   A_3126_BTE05.Par.OutDelayTime := 0;
   A_3126_BTE05.Par.Spare66 := 0;
   A_3126_BTE06.StCode := 0;
   A_3126_BTE06.InMonLL := FALSE;
   A_3126_BTE06.InMonL := FALSE;
   A_3126_BTE06.InMonMid := FALSE;
   A_3126_BTE06.InMonH := FALSE;
   A_3126_BTE06.InMonHH := FALSE;
   A_3126_BTE06.spare0205 := FALSE;
   A_3126_BTE06.InpFaultAI := FALSE;
   A_3126_BTE06.InpFaultDev := FALSE;
   A_3126_BTE06.InHWStop := FALSE;
   A_3126_BTE06.InDPFault := FALSE;
   A_3126_BTE06.InDisable := FALSE;
   A_3126_BTE06.CmdFaultReset := FALSE;
   A_3126_BTE06.InLocal := FALSE;
   A_3126_BTE06.spare0305 := FALSE;
   A_3126_BTE06.InReport := FALSE;
   A_3126_BTE06.spare0307 := FALSE;
   A_3126_BTE06.OutLL := FALSE;
   A_3126_BTE06.OutL := FALSE;
   A_3126_BTE06.OutH := FALSE;
   A_3126_BTE06.OutHH := FALSE;
   A_3126_BTE06.OutOverflow := FALSE;
   A_3126_BTE06.spare0405 := FALSE;
   A_3126_BTE06.OutFaultAI := FALSE;
   A_3126_BTE06.spare0407 := FALSE;
   A_3126_BTE06.StLL := FALSE;
   A_3126_BTE06.StL := FALSE;
   A_3126_BTE06.StMid := FALSE;
   A_3126_BTE06.StH := FALSE;
   A_3126_BTE06.StHH := FALSE;
   A_3126_BTE06.StFaultAI := FALSE;
   A_3126_BTE06.OutWarning := FALSE;
   A_3126_BTE06.OutFaulted := FALSE;
   A_3126_BTE06.InpValue := 0;
   A_3126_BTE06.OutValuePc := 0;
   A_3126_BTE06.OutValueUnits := L#0;
   A_3126_BTE06.Msg.WarningDoneLL := FALSE;
   A_3126_BTE06.Msg.WarningDoneL := FALSE;
   A_3126_BTE06.Msg.WarningDoneMid := FALSE;
   A_3126_BTE06.Msg.WarningDoneH := FALSE;
   A_3126_BTE06.Msg.WarningDoneHH := FALSE;
   A_3126_BTE06.Msg.FaultDoneLL := FALSE;
   A_3126_BTE06.Msg.FaultDoneL := FALSE;
   A_3126_BTE06.Msg.FaultDoneMid := FALSE;
   A_3126_BTE06.Msg.FaultDoneH := FALSE;
   A_3126_BTE06.Msg.FaultDoneHH := FALSE;
   A_3126_BTE06.Msg.FaultDoneDev := FALSE;
   A_3126_BTE06.Msg.FaultDoneAI := FALSE;
   A_3126_BTE06.OutAlarmNrLog := 0;
   A_3126_BTE06.Par.ParObjectNo := 27118;
   A_3126_BTE06.Par.ParMsgType := 7252;
   A_3126_BTE06.Par.ParHornCode := 10;
   A_3126_BTE06.Par.ParLogOff := FALSE;
   A_3126_BTE06.Par.ParSpare0401 := FALSE;
   A_3126_BTE06.Par.ParValueByUser := FALSE;
   A_3126_BTE06.Par.ParLimitsPc := TRUE;
   A_3126_BTE06.Par.ParWago := FALSE;
   A_3126_BTE06.Par.ParNoHornByWarning := FALSE;
   A_3126_BTE06.Par.ParWarningLL := FALSE;
   A_3126_BTE06.Par.ParWarningL := FALSE;
   A_3126_BTE06.Par.ParWarningMid := FALSE;
   A_3126_BTE06.Par.ParWarningH := TRUE;
   A_3126_BTE06.Par.ParWarningHH := FALSE;
   A_3126_BTE06.Par.ParPreAlarmLL := FALSE;
   A_3126_BTE06.Par.ParPreAlarmL := FALSE;
   A_3126_BTE06.Par.ParPreAlarmMid := FALSE;
   A_3126_BTE06.Par.ParPreAlarmH := FALSE;
   A_3126_BTE06.Par.ParPreAlarmHH := FALSE;
   A_3126_BTE06.Par.ParUnitsByZeroDigit := L#0;
   A_3126_BTE06.Par.ParUnitsByMaxDigit := L#27384;
   A_3126_BTE06.Par.ParUnitsBy100Pc := L#10000;
   A_3126_BTE06.Par.ParLimitLL := L#0;
   A_3126_BTE06.Par.ParLimitL := L#2000;
   A_3126_BTE06.Par.ParLimitH := L#8000;
   A_3126_BTE06.Par.ParLimitHH := L#10000;
   A_3126_BTE06.Par.ParMonTimeLL := 0;
   A_3126_BTE06.Par.ParMonTimeL := 0;
   A_3126_BTE06.Par.ParMonTimeMid := 0;
   A_3126_BTE06.Par.ParMonTimeH := 600;
   A_3126_BTE06.Par.ParMonTimeHH := 0;
   A_3126_BTE06.Par.ParDelayTimeDown := 10;
   A_3126_BTE06.Par.ParDelayTimeUp := 10;
   A_3126_BTE06.Par.ParDelayTime := 30;
   A_3126_BTE06.Par.OutMonTimeLL := 0;
   A_3126_BTE06.Par.OutMonTimeL := 0;
   A_3126_BTE06.Par.OutMonTimeMid := 0;
   A_3126_BTE06.Par.OutMonTimeH := 0;
   A_3126_BTE06.Par.OutMonTimeHH := 0;
   A_3126_BTE06.Par.OutDelayTimeDown := 0;
   A_3126_BTE06.Par.OutDelayTimeUp := 0;
   A_3126_BTE06.Par.OutDelayTime := 0;
   A_3126_BTE06.Par.Spare66 := 0;
   A_3126_MXZ01MA.Ma.StCode := 0;
   A_3126_MXZ01MA.Ma.InEnableRev := FALSE;
   A_3126_MXZ01MA.Ma.InEnableFwd := FALSE;
   A_3126_MXZ01MA.Ma.InOverrideHLOutlet := FALSE;
   A_3126_MXZ01MA.Ma.spare0203 := FALSE;
   A_3126_MXZ01MA.Ma.OutEdgeFaultReset := FALSE;
   A_3126_MXZ01MA.Ma.OutFaultResetFcttst := FALSE;
   A_3126_MXZ01MA.Ma.InpControlEBM := FALSE;
   A_3126_MXZ01MA.Ma.InpLocked := FALSE;
   A_3126_MXZ01MA.Ma.CmdOff := FALSE;
   A_3126_MXZ01MA.Ma.CmdOn := FALSE;
   A_3126_MXZ01MA.Ma.CmdNext := FALSE;
   A_3126_MXZ01MA.Ma.CmdFaultReset := FALSE;
   A_3126_MXZ01MA.Ma.InLocal := FALSE;
   A_3126_MXZ01MA.Ma.InManual := FALSE;
   A_3126_MXZ01MA.Ma.CmdTestEBM := FALSE;
   A_3126_MXZ01MA.Ma.InSeqStop := FALSE;
   A_3126_MXZ01MA.Ma.OutWarning := FALSE;
   A_3126_MXZ01MA.Ma.InfBMTopOk := FALSE;
   A_3126_MXZ01MA.Ma.InfBMBottomOk := FALSE;
   A_3126_MXZ01MA.Ma.InfSMOk := FALSE;
   A_3126_MXZ01MA.Ma.OutpFcttst_BM_Top := FALSE;
   A_3126_MXZ01MA.Ma.OutpFcttst_BM_Bottom := FALSE;
   A_3126_MXZ01MA.Ma.OutpFcttst_SM := FALSE;
   A_3126_MXZ01MA.Ma.OutpFaultReset := FALSE;
   A_3126_MXZ01MA.Ma.StStopped := FALSE;
   A_3126_MXZ01MA.Ma.StStarting := FALSE;
   A_3126_MXZ01MA.Ma.StStartedFwd := FALSE;
   A_3126_MXZ01MA.Ma.StStopping := FALSE;
   A_3126_MXZ01MA.Ma.StFault := FALSE;
   A_3126_MXZ01MA.Ma.StStartedRev := FALSE;
   A_3126_MXZ01MA.Ma.StLocked := FALSE;
   A_3126_MXZ01MA.Ma.OutTestTime := 0;
   A_3126_MXZ01MA.Ma.Par.ParObjectNo := 27119;
   A_3126_MXZ01MA.Ma.Par.ParWithMon1 := TRUE;
   A_3126_MXZ01MA.Ma.Par.ParWithMon3 := FALSE;
   A_3126_MXZ01MA.Ma.Par.ParWithMon4 := TRUE;
   A_3126_MXZ01MA.Ma.Par.ParWithMon5 := FALSE;
   A_3126_MXZ01MA.Ma.Par.ParWithMon6 := FALSE;
   A_3126_MXZ01MA.Ma.Par.ParMon1IsHL := FALSE;
   A_3126_MXZ01MA.Ma.Par.ParMon1IsLS := TRUE;
   A_3126_MXZ01MA.Ma.Par.ParMon1StopByFault := TRUE;
   A_3126_MXZ01MA.Ma.Par.ParMon2IsLS := FALSE;
   A_3126_MXZ01MA.Ma.Par.ParMon3IsLS := FALSE;
   A_3126_MXZ01MA.Ma.Par.ParMon4AsWarning := FALSE;
   A_3126_MXZ01MA.Ma.Par.ParMon4StopByFault := FALSE;
   A_3126_MXZ01MA.Ma.Par.ParMon4IsLS := FALSE;
   A_3126_MXZ01MA.Ma.Par.ParEBM := FALSE;
   A_3126_MXZ01MA.Ma.Par.ParMon4IsSM := TRUE;
   A_3126_MXZ01MA.A_3126_KCU04.StCode := 0;
   A_3126_MXZ01MA.A_3126_KCU04.InMonTrue := FALSE;
   A_3126_MXZ01MA.A_3126_KCU04.InMonFalse := FALSE;
   A_3126_MXZ01MA.A_3126_KCU04.InPreAlarmTrue := FALSE;
   A_3126_MXZ01MA.A_3126_KCU04.InPreAlarmFalse := FALSE;
   A_3126_MXZ01MA.A_3126_KCU04.InStopTrueTime := FALSE;
   A_3126_MXZ01MA.A_3126_KCU04.InStopFalseTime := FALSE;
   A_3126_MXZ01MA.A_3126_KCU04.InpTrue := FALSE;
   A_3126_MXZ01MA.A_3126_KCU04.InpFaultDev := FALSE;
   A_3126_MXZ01MA.A_3126_KCU04.CmdRstTrueTime := FALSE;
   A_3126_MXZ01MA.A_3126_KCU04.CmdRstFalseTime := FALSE;
   A_3126_MXZ01MA.A_3126_KCU04.CmdRunTimeoutTime := FALSE;
   A_3126_MXZ01MA.A_3126_KCU04.CmdFaultReset := FALSE;
   A_3126_MXZ01MA.A_3126_KCU04.InLocal := FALSE;
   A_3126_MXZ01MA.A_3126_KCU04.spare0305 := FALSE;
   A_3126_MXZ01MA.A_3126_KCU04.InReport := FALSE;
   A_3126_MXZ01MA.A_3126_KCU04.OutTimeoutTime := FALSE;
   A_3126_MXZ01MA.A_3126_KCU04.InHWStop := FALSE;
   A_3126_MXZ01MA.A_3126_KCU04.InDPFault := FALSE;
   A_3126_MXZ01MA.A_3126_KCU04.OutPreAlarmTrue := FALSE;
   A_3126_MXZ01MA.A_3126_KCU04.OutPreAlarmFalse := FALSE;
   A_3126_MXZ01MA.A_3126_KCU04.OutFlagPos := FALSE;
   A_3126_MXZ01MA.A_3126_KCU04.OutFlagNeg := FALSE;
   A_3126_MXZ01MA.A_3126_KCU04.OutpFaultReset := FALSE;
   A_3126_MXZ01MA.A_3126_KCU04.OutTrue := FALSE;
   A_3126_MXZ01MA.A_3126_KCU04.StFalse := FALSE;
   A_3126_MXZ01MA.A_3126_KCU04.StCtoTrue := FALSE;
   A_3126_MXZ01MA.A_3126_KCU04.StTrue := FALSE;
   A_3126_MXZ01MA.A_3126_KCU04.StCtoFalse := FALSE;
   A_3126_MXZ01MA.A_3126_KCU04.StFault := FALSE;
   A_3126_MXZ01MA.A_3126_KCU04.OutAlarmNrLog := 0;
   A_3126_MXZ01MA.A_3126_KCU04.Par.ParObjectNo := 27120;
   A_3126_MXZ01MA.A_3126_KCU04.Par.ParMsgType := 7154;
   A_3126_MXZ01MA.A_3126_KCU04.Par.ParHornCode := 10;
   A_3126_MXZ01MA.A_3126_KCU04.Par.ParLogOff := FALSE;
   A_3126_MXZ01MA.A_3126_KCU04.Par.spare0401 := FALSE;
   A_3126_MXZ01MA.A_3126_KCU04.Par.Par2WorkingCond := FALSE;
   A_3126_MXZ01MA.A_3126_KCU04.Par.ParFaultRetry := FALSE;
   A_3126_MXZ01MA.A_3126_KCU04.Par.ParBinLevel := FALSE;
   A_3126_MXZ01MA.A_3126_KCU04.Par.ParDelayChange := 20;
   A_3126_MXZ01MA.A_3126_KCU04.Par.ParDelayTrue := 10;
   A_3126_MXZ01MA.A_3126_KCU04.Par.ParDelayFalse := 0;
   A_3126_MXZ01MA.A_3126_KCU04.Par.ParTimeoutTrue := 0;
   A_3126_MXZ01MA.A_3126_KCU04.Par.ParTimeoutFalse := 0;
   A_3126_MXZ01MA.A_3126_KCU04.Par.OutMonTime := 0;
   A_3126_MXZ01MA.A_3126_KCU04.Par.OutTransitionTime := 0;
   A_3126_MXZ01MA.A_3126_KCU04.Par.OutMonTrue := FALSE;
   A_3126_MXZ01MA.A_3126_KCU04.Par.OutMonFalse := FALSE;
   A_3126_MXZ01MA.A_3126_KCU04.Par.OutFlagFaultDev := FALSE;
   A_3126_MXZ01MA.A_3126_KCU04.Par.OutDelayTime := 0;
   A_3126_MXZ01MA.Mon2.StCode := 0;
   A_3126_MXZ01MA.Mon2.InMonTrue := FALSE;
   A_3126_MXZ01MA.Mon2.InMonFalse := FALSE;
   A_3126_MXZ01MA.Mon2.InPreAlarmTrue := FALSE;
   A_3126_MXZ01MA.Mon2.InPreAlarmFalse := FALSE;
   A_3126_MXZ01MA.Mon2.InStopTrueTime := FALSE;
   A_3126_MXZ01MA.Mon2.InStopFalseTime := FALSE;
   A_3126_MXZ01MA.Mon2.InpTrue := FALSE;
   A_3126_MXZ01MA.Mon2.InpFaultDev := FALSE;
   A_3126_MXZ01MA.Mon2.CmdRstTrueTime := FALSE;
   A_3126_MXZ01MA.Mon2.CmdRstFalseTime := FALSE;
   A_3126_MXZ01MA.Mon2.CmdRunTimeoutTime := FALSE;
   A_3126_MXZ01MA.Mon2.CmdFaultReset := FALSE;
   A_3126_MXZ01MA.Mon2.InLocal := FALSE;
   A_3126_MXZ01MA.Mon2.spare0305 := FALSE;
   A_3126_MXZ01MA.Mon2.InReport := FALSE;
   A_3126_MXZ01MA.Mon2.OutTimeoutTime := FALSE;
   A_3126_MXZ01MA.Mon2.InHWStop := FALSE;
   A_3126_MXZ01MA.Mon2.InDPFault := FALSE;
   A_3126_MXZ01MA.Mon2.OutPreAlarmTrue := FALSE;
   A_3126_MXZ01MA.Mon2.OutPreAlarmFalse := FALSE;
   A_3126_MXZ01MA.Mon2.OutFlagPos := FALSE;
   A_3126_MXZ01MA.Mon2.OutFlagNeg := FALSE;
   A_3126_MXZ01MA.Mon2.OutpFaultReset := FALSE;
   A_3126_MXZ01MA.Mon2.OutTrue := FALSE;
   A_3126_MXZ01MA.Mon2.StFalse := FALSE;
   A_3126_MXZ01MA.Mon2.StCtoTrue := FALSE;
   A_3126_MXZ01MA.Mon2.StTrue := FALSE;
   A_3126_MXZ01MA.Mon2.StCtoFalse := FALSE;
   A_3126_MXZ01MA.Mon2.StFault := FALSE;
   A_3126_MXZ01MA.Mon2.OutAlarmNrLog := 0;
   A_3126_MXZ01MA.Mon2.Par.ParObjectNo := 0;
   A_3126_MXZ01MA.Mon2.Par.ParMsgType := 0;
   A_3126_MXZ01MA.Mon2.Par.ParHornCode := 0;
   A_3126_MXZ01MA.Mon2.Par.ParLogOff := FALSE;
   A_3126_MXZ01MA.Mon2.Par.spare0401 := FALSE;
   A_3126_MXZ01MA.Mon2.Par.Par2WorkingCond := FALSE;
   A_3126_MXZ01MA.Mon2.Par.ParFaultRetry := FALSE;
   A_3126_MXZ01MA.Mon2.Par.ParBinLevel := FALSE;
   A_3126_MXZ01MA.Mon2.Par.ParDelayChange := 0;
   A_3126_MXZ01MA.Mon2.Par.ParDelayTrue := 0;
   A_3126_MXZ01MA.Mon2.Par.ParDelayFalse := 0;
   A_3126_MXZ01MA.Mon2.Par.ParTimeoutTrue := 0;
   A_3126_MXZ01MA.Mon2.Par.ParTimeoutFalse := 0;
   A_3126_MXZ01MA.Mon2.Par.OutMonTime := 0;
   A_3126_MXZ01MA.Mon2.Par.OutTransitionTime := 0;
   A_3126_MXZ01MA.Mon2.Par.OutMonTrue := FALSE;
   A_3126_MXZ01MA.Mon2.Par.OutMonFalse := FALSE;
   A_3126_MXZ01MA.Mon2.Par.OutFlagFaultDev := FALSE;
   A_3126_MXZ01MA.Mon2.Par.OutDelayTime := 0;
   A_3126_MXZ01MA.Mon3.StCode := 0;
   A_3126_MXZ01MA.Mon3.InMonTrue := FALSE;
   A_3126_MXZ01MA.Mon3.InMonFalse := FALSE;
   A_3126_MXZ01MA.Mon3.InPreAlarmTrue := FALSE;
   A_3126_MXZ01MA.Mon3.InPreAlarmFalse := FALSE;
   A_3126_MXZ01MA.Mon3.InStopTrueTime := FALSE;
   A_3126_MXZ01MA.Mon3.InStopFalseTime := FALSE;
   A_3126_MXZ01MA.Mon3.InpTrue := FALSE;
   A_3126_MXZ01MA.Mon3.InpFaultDev := FALSE;
   A_3126_MXZ01MA.Mon3.CmdRstTrueTime := FALSE;
   A_3126_MXZ01MA.Mon3.CmdRstFalseTime := FALSE;
   A_3126_MXZ01MA.Mon3.CmdRunTimeoutTime := FALSE;
   A_3126_MXZ01MA.Mon3.CmdFaultReset := FALSE;
   A_3126_MXZ01MA.Mon3.InLocal := FALSE;
   A_3126_MXZ01MA.Mon3.spare0305 := FALSE;
   A_3126_MXZ01MA.Mon3.InReport := FALSE;
   A_3126_MXZ01MA.Mon3.OutTimeoutTime := FALSE;
   A_3126_MXZ01MA.Mon3.InHWStop := FALSE;
   A_3126_MXZ01MA.Mon3.InDPFault := FALSE;
   A_3126_MXZ01MA.Mon3.OutPreAlarmTrue := FALSE;
   A_3126_MXZ01MA.Mon3.OutPreAlarmFalse := FALSE;
   A_3126_MXZ01MA.Mon3.OutFlagPos := FALSE;
   A_3126_MXZ01MA.Mon3.OutFlagNeg := FALSE;
   A_3126_MXZ01MA.Mon3.OutpFaultReset := FALSE;
   A_3126_MXZ01MA.Mon3.OutTrue := FALSE;
   A_3126_MXZ01MA.Mon3.StFalse := FALSE;
   A_3126_MXZ01MA.Mon3.StCtoTrue := FALSE;
   A_3126_MXZ01MA.Mon3.StTrue := FALSE;
   A_3126_MXZ01MA.Mon3.StCtoFalse := FALSE;
   A_3126_MXZ01MA.Mon3.StFault := FALSE;
   A_3126_MXZ01MA.Mon3.OutAlarmNrLog := 0;
   A_3126_MXZ01MA.Mon3.Par.ParObjectNo := 0;
   A_3126_MXZ01MA.Mon3.Par.ParMsgType := 0;
   A_3126_MXZ01MA.Mon3.Par.ParHornCode := 0;
   A_3126_MXZ01MA.Mon3.Par.ParLogOff := FALSE;
   A_3126_MXZ01MA.Mon3.Par.spare0401 := FALSE;
   A_3126_MXZ01MA.Mon3.Par.Par2WorkingCond := FALSE;
   A_3126_MXZ01MA.Mon3.Par.ParFaultRetry := FALSE;
   A_3126_MXZ01MA.Mon3.Par.ParBinLevel := FALSE;
   A_3126_MXZ01MA.Mon3.Par.ParDelayChange := 0;
   A_3126_MXZ01MA.Mon3.Par.ParDelayTrue := 0;
   A_3126_MXZ01MA.Mon3.Par.ParDelayFalse := 0;
   A_3126_MXZ01MA.Mon3.Par.ParTimeoutTrue := 0;
   A_3126_MXZ01MA.Mon3.Par.ParTimeoutFalse := 0;
   A_3126_MXZ01MA.Mon3.Par.OutMonTime := 0;
   A_3126_MXZ01MA.Mon3.Par.OutTransitionTime := 0;
   A_3126_MXZ01MA.Mon3.Par.OutMonTrue := FALSE;
   A_3126_MXZ01MA.Mon3.Par.OutMonFalse := FALSE;
   A_3126_MXZ01MA.Mon3.Par.OutFlagFaultDev := FALSE;
   A_3126_MXZ01MA.Mon3.Par.OutDelayTime := 0;
   A_3126_MXZ01MA.A_3126_BSA07.StCode := 0;
   A_3126_MXZ01MA.A_3126_BSA07.InMonTrue := FALSE;
   A_3126_MXZ01MA.A_3126_BSA07.InMonFalse := FALSE;
   A_3126_MXZ01MA.A_3126_BSA07.InPreAlarmTrue := FALSE;
   A_3126_MXZ01MA.A_3126_BSA07.InPreAlarmFalse := FALSE;
   A_3126_MXZ01MA.A_3126_BSA07.InStopTrueTime := FALSE;
   A_3126_MXZ01MA.A_3126_BSA07.InStopFalseTime := FALSE;
   A_3126_MXZ01MA.A_3126_BSA07.InpTrue := FALSE;
   A_3126_MXZ01MA.A_3126_BSA07.InpFaultDev := FALSE;
   A_3126_MXZ01MA.A_3126_BSA07.CmdRstTrueTime := FALSE;
   A_3126_MXZ01MA.A_3126_BSA07.CmdRstFalseTime := FALSE;
   A_3126_MXZ01MA.A_3126_BSA07.CmdRunTimeoutTime := FALSE;
   A_3126_MXZ01MA.A_3126_BSA07.CmdFaultReset := FALSE;
   A_3126_MXZ01MA.A_3126_BSA07.InLocal := FALSE;
   A_3126_MXZ01MA.A_3126_BSA07.spare0305 := FALSE;
   A_3126_MXZ01MA.A_3126_BSA07.InReport := FALSE;
   A_3126_MXZ01MA.A_3126_BSA07.OutTimeoutTime := FALSE;
   A_3126_MXZ01MA.A_3126_BSA07.InHWStop := FALSE;
   A_3126_MXZ01MA.A_3126_BSA07.InDPFault := FALSE;
   A_3126_MXZ01MA.A_3126_BSA07.OutPreAlarmTrue := FALSE;
   A_3126_MXZ01MA.A_3126_BSA07.OutPreAlarmFalse := FALSE;
   A_3126_MXZ01MA.A_3126_BSA07.OutFlagPos := FALSE;
   A_3126_MXZ01MA.A_3126_BSA07.OutFlagNeg := FALSE;
   A_3126_MXZ01MA.A_3126_BSA07.OutpFaultReset := FALSE;
   A_3126_MXZ01MA.A_3126_BSA07.OutTrue := FALSE;
   A_3126_MXZ01MA.A_3126_BSA07.StFalse := FALSE;
   A_3126_MXZ01MA.A_3126_BSA07.StCtoTrue := FALSE;
   A_3126_MXZ01MA.A_3126_BSA07.StTrue := FALSE;
   A_3126_MXZ01MA.A_3126_BSA07.StCtoFalse := FALSE;
   A_3126_MXZ01MA.A_3126_BSA07.StFault := FALSE;
   A_3126_MXZ01MA.A_3126_BSA07.OutAlarmNrLog := 0;
   A_3126_MXZ01MA.A_3126_BSA07.Par.ParObjectNo := 27134;
   A_3126_MXZ01MA.A_3126_BSA07.Par.ParMsgType := 7135;
   A_3126_MXZ01MA.A_3126_BSA07.Par.ParHornCode := 0;
   A_3126_MXZ01MA.A_3126_BSA07.Par.ParLogOff := FALSE;
   A_3126_MXZ01MA.A_3126_BSA07.Par.spare0401 := FALSE;
   A_3126_MXZ01MA.A_3126_BSA07.Par.Par2WorkingCond := TRUE;
   A_3126_MXZ01MA.A_3126_BSA07.Par.ParFaultRetry := FALSE;
   A_3126_MXZ01MA.A_3126_BSA07.Par.ParBinLevel := FALSE;
   A_3126_MXZ01MA.A_3126_BSA07.Par.ParDelayChange := 0;
   A_3126_MXZ01MA.A_3126_BSA07.Par.ParDelayTrue := 200;
   A_3126_MXZ01MA.A_3126_BSA07.Par.ParDelayFalse := 0;
   A_3126_MXZ01MA.A_3126_BSA07.Par.ParTimeoutTrue := 50;
   A_3126_MXZ01MA.A_3126_BSA07.Par.ParTimeoutFalse := 0;
   A_3126_MXZ01MA.A_3126_BSA07.Par.OutMonTime := 0;
   A_3126_MXZ01MA.A_3126_BSA07.Par.OutTransitionTime := 0;
   A_3126_MXZ01MA.A_3126_BSA07.Par.OutMonTrue := FALSE;
   A_3126_MXZ01MA.A_3126_BSA07.Par.OutMonFalse := FALSE;
   A_3126_MXZ01MA.A_3126_BSA07.Par.OutFlagFaultDev := FALSE;
   A_3126_MXZ01MA.A_3126_BSA07.Par.OutDelayTime := 0;
   A_3126_MXZ01MA.Mon5.StCode := 0;
   A_3126_MXZ01MA.Mon5.InMonTrue := FALSE;
   A_3126_MXZ01MA.Mon5.InMonFalse := FALSE;
   A_3126_MXZ01MA.Mon5.InPreAlarmTrue := FALSE;
   A_3126_MXZ01MA.Mon5.InPreAlarmFalse := FALSE;
   A_3126_MXZ01MA.Mon5.InStopTrueTime := FALSE;
   A_3126_MXZ01MA.Mon5.InStopFalseTime := FALSE;
   A_3126_MXZ01MA.Mon5.InpTrue := FALSE;
   A_3126_MXZ01MA.Mon5.InpFaultDev := FALSE;
   A_3126_MXZ01MA.Mon5.CmdRstTrueTime := FALSE;
   A_3126_MXZ01MA.Mon5.CmdRstFalseTime := FALSE;
   A_3126_MXZ01MA.Mon5.CmdRunTimeoutTime := FALSE;
   A_3126_MXZ01MA.Mon5.CmdFaultReset := FALSE;
   A_3126_MXZ01MA.Mon5.InLocal := FALSE;
   A_3126_MXZ01MA.Mon5.spare0305 := FALSE;
   A_3126_MXZ01MA.Mon5.InReport := FALSE;
   A_3126_MXZ01MA.Mon5.OutTimeoutTime := FALSE;
   A_3126_MXZ01MA.Mon5.InHWStop := FALSE;
   A_3126_MXZ01MA.Mon5.InDPFault := FALSE;
   A_3126_MXZ01MA.Mon5.OutPreAlarmTrue := FALSE;
   A_3126_MXZ01MA.Mon5.OutPreAlarmFalse := FALSE;
   A_3126_MXZ01MA.Mon5.OutFlagPos := FALSE;
   A_3126_MXZ01MA.Mon5.OutFlagNeg := FALSE;
   A_3126_MXZ01MA.Mon5.OutpFaultReset := FALSE;
   A_3126_MXZ01MA.Mon5.OutTrue := FALSE;
   A_3126_MXZ01MA.Mon5.StFalse := FALSE;
   A_3126_MXZ01MA.Mon5.StCtoTrue := FALSE;
   A_3126_MXZ01MA.Mon5.StTrue := FALSE;
   A_3126_MXZ01MA.Mon5.StCtoFalse := FALSE;
   A_3126_MXZ01MA.Mon5.StFault := FALSE;
   A_3126_MXZ01MA.Mon5.OutAlarmNrLog := 0;
   A_3126_MXZ01MA.Mon5.Par.ParObjectNo := 0;
   A_3126_MXZ01MA.Mon5.Par.ParMsgType := 0;
   A_3126_MXZ01MA.Mon5.Par.ParHornCode := 0;
   A_3126_MXZ01MA.Mon5.Par.ParLogOff := FALSE;
   A_3126_MXZ01MA.Mon5.Par.spare0401 := FALSE;
   A_3126_MXZ01MA.Mon5.Par.Par2WorkingCond := FALSE;
   A_3126_MXZ01MA.Mon5.Par.ParFaultRetry := FALSE;
   A_3126_MXZ01MA.Mon5.Par.ParBinLevel := FALSE;
   A_3126_MXZ01MA.Mon5.Par.ParDelayChange := 0;
   A_3126_MXZ01MA.Mon5.Par.ParDelayTrue := 0;
   A_3126_MXZ01MA.Mon5.Par.ParDelayFalse := 0;
   A_3126_MXZ01MA.Mon5.Par.ParTimeoutTrue := 0;
   A_3126_MXZ01MA.Mon5.Par.ParTimeoutFalse := 0;
   A_3126_MXZ01MA.Mon5.Par.OutMonTime := 0;
   A_3126_MXZ01MA.Mon5.Par.OutTransitionTime := 0;
   A_3126_MXZ01MA.Mon5.Par.OutMonTrue := FALSE;
   A_3126_MXZ01MA.Mon5.Par.OutMonFalse := FALSE;
   A_3126_MXZ01MA.Mon5.Par.OutFlagFaultDev := FALSE;
   A_3126_MXZ01MA.Mon5.Par.OutDelayTime := 0;
   A_3126_MXZ01MA.Mon6.StCode := 0;
   A_3126_MXZ01MA.Mon6.InMonTrue := FALSE;
   A_3126_MXZ01MA.Mon6.InMonFalse := FALSE;
   A_3126_MXZ01MA.Mon6.InPreAlarmTrue := FALSE;
   A_3126_MXZ01MA.Mon6.InPreAlarmFalse := FALSE;
   A_3126_MXZ01MA.Mon6.InStopTrueTime := FALSE;
   A_3126_MXZ01MA.Mon6.InStopFalseTime := FALSE;
   A_3126_MXZ01MA.Mon6.InpTrue := FALSE;
   A_3126_MXZ01MA.Mon6.InpFaultDev := FALSE;
   A_3126_MXZ01MA.Mon6.CmdRstTrueTime := FALSE;
   A_3126_MXZ01MA.Mon6.CmdRstFalseTime := FALSE;
   A_3126_MXZ01MA.Mon6.CmdRunTimeoutTime := FALSE;
   A_3126_MXZ01MA.Mon6.CmdFaultReset := FALSE;
   A_3126_MXZ01MA.Mon6.InLocal := FALSE;
   A_3126_MXZ01MA.Mon6.spare0305 := FALSE;
   A_3126_MXZ01MA.Mon6.InReport := FALSE;
   A_3126_MXZ01MA.Mon6.OutTimeoutTime := FALSE;
   A_3126_MXZ01MA.Mon6.InHWStop := FALSE;
   A_3126_MXZ01MA.Mon6.InDPFault := FALSE;
   A_3126_MXZ01MA.Mon6.OutPreAlarmTrue := FALSE;
   A_3126_MXZ01MA.Mon6.OutPreAlarmFalse := FALSE;
   A_3126_MXZ01MA.Mon6.OutFlagPos := FALSE;
   A_3126_MXZ01MA.Mon6.OutFlagNeg := FALSE;
   A_3126_MXZ01MA.Mon6.OutpFaultReset := FALSE;
   A_3126_MXZ01MA.Mon6.OutTrue := FALSE;
   A_3126_MXZ01MA.Mon6.StFalse := FALSE;
   A_3126_MXZ01MA.Mon6.StCtoTrue := FALSE;
   A_3126_MXZ01MA.Mon6.StTrue := FALSE;
   A_3126_MXZ01MA.Mon6.StCtoFalse := FALSE;
   A_3126_MXZ01MA.Mon6.StFault := FALSE;
   A_3126_MXZ01MA.Mon6.OutAlarmNrLog := 0;
   A_3126_MXZ01MA.Mon6.Par.ParObjectNo := 0;
   A_3126_MXZ01MA.Mon6.Par.ParMsgType := 0;
   A_3126_MXZ01MA.Mon6.Par.ParHornCode := 0;
   A_3126_MXZ01MA.Mon6.Par.ParLogOff := FALSE;
   A_3126_MXZ01MA.Mon6.Par.spare0401 := FALSE;
   A_3126_MXZ01MA.Mon6.Par.Par2WorkingCond := FALSE;
   A_3126_MXZ01MA.Mon6.Par.ParFaultRetry := FALSE;
   A_3126_MXZ01MA.Mon6.Par.ParBinLevel := FALSE;
   A_3126_MXZ01MA.Mon6.Par.ParDelayChange := 0;
   A_3126_MXZ01MA.Mon6.Par.ParDelayTrue := 0;
   A_3126_MXZ01MA.Mon6.Par.ParDelayFalse := 0;
   A_3126_MXZ01MA.Mon6.Par.ParTimeoutTrue := 0;
   A_3126_MXZ01MA.Mon6.Par.ParTimeoutFalse := 0;
   A_3126_MXZ01MA.Mon6.Par.OutMonTime := 0;
   A_3126_MXZ01MA.Mon6.Par.OutTransitionTime := 0;
   A_3126_MXZ01MA.Mon6.Par.OutMonTrue := FALSE;
   A_3126_MXZ01MA.Mon6.Par.OutMonFalse := FALSE;
   A_3126_MXZ01MA.Mon6.Par.OutFlagFaultDev := FALSE;
   A_3126_MXZ01MA.Mon6.Par.OutDelayTime := 0;
   A_3126_MXZ01MA.A_3126_MXZ01.StCode := 0;
   A_3126_MXZ01MA.A_3126_MXZ01.InEnableRev := FALSE;
   A_3126_MXZ01MA.A_3126_MXZ01.InEnableFwd := FALSE;
   A_3126_MXZ01MA.A_3126_MXZ01.InSlow := FALSE;
   A_3126_MXZ01MA.A_3126_MXZ01.InpRunSlow := FALSE;
   A_3126_MXZ01MA.A_3126_MXZ01.InpRunFast := FALSE;
   A_3126_MXZ01MA.A_3126_MXZ01.InpRunRev := FALSE;
   A_3126_MXZ01MA.A_3126_MXZ01.InpRunFwd := FALSE;
   A_3126_MXZ01MA.A_3126_MXZ01.InpFaultDev := FALSE;
   A_3126_MXZ01MA.A_3126_MXZ01.CmdOff := FALSE;
   A_3126_MXZ01MA.A_3126_MXZ01.CmdOn := FALSE;
   A_3126_MXZ01MA.A_3126_MXZ01.CmdNext := FALSE;
   A_3126_MXZ01MA.A_3126_MXZ01.CmdFaultReset := FALSE;
   A_3126_MXZ01MA.A_3126_MXZ01.InLocal := FALSE;
   A_3126_MXZ01MA.A_3126_MXZ01.InManual := FALSE;
   A_3126_MXZ01MA.A_3126_MXZ01.InReport := FALSE;
   A_3126_MXZ01MA.A_3126_MXZ01.InSeqStop := FALSE;
   A_3126_MXZ01MA.A_3126_MXZ01.InHWStop := FALSE;
   A_3126_MXZ01MA.A_3126_MXZ01.InDPFault := FALSE;
   A_3126_MXZ01MA.A_3126_MXZ01.OutIdling := FALSE;
   A_3126_MXZ01MA.A_3126_MXZ01.OutpRunSlow := FALSE;
   A_3126_MXZ01MA.A_3126_MXZ01.OutpRunFast := FALSE;
   A_3126_MXZ01MA.A_3126_MXZ01.OutpRunRev := FALSE;
   A_3126_MXZ01MA.A_3126_MXZ01.OutpRunFwd := FALSE;
   A_3126_MXZ01MA.A_3126_MXZ01.OutpFaultReset := FALSE;
   A_3126_MXZ01MA.A_3126_MXZ01.StStopped := FALSE;
   A_3126_MXZ01MA.A_3126_MXZ01.StStarting := FALSE;
   A_3126_MXZ01MA.A_3126_MXZ01.StStartedFwd := FALSE;
   A_3126_MXZ01MA.A_3126_MXZ01.StStopping := FALSE;
   A_3126_MXZ01MA.A_3126_MXZ01.StFault := FALSE;
   A_3126_MXZ01MA.A_3126_MXZ01.StStartedRev := FALSE;
   A_3126_MXZ01MA.A_3126_MXZ01.InOutManSlow := FALSE;
   A_3126_MXZ01MA.A_3126_MXZ01.InOutManRev := FALSE;
   A_3126_MXZ01MA.A_3126_MXZ01.OutAlarmNrLog := 0;
   A_3126_MXZ01MA.A_3126_MXZ01.Par.ParObjectNo := 27122;
   A_3126_MXZ01MA.A_3126_MXZ01.Par.ParMsgType := 7053;
   A_3126_MXZ01MA.A_3126_MXZ01.Par.ParHornCode := 10;
   A_3126_MXZ01MA.A_3126_MXZ01.Par.ParLogOff := FALSE;
   A_3126_MXZ01MA.A_3126_MXZ01.Par.ParManual := TRUE;
   A_3126_MXZ01MA.A_3126_MXZ01.Par.ParRestartDelay := FALSE;
   A_3126_MXZ01MA.A_3126_MXZ01.Par.Par2Speed := FALSE;
   A_3126_MXZ01MA.A_3126_MXZ01.Par.ParHeavyStartup := FALSE;
   A_3126_MXZ01MA.A_3126_MXZ01.Par.spare45 := FALSE;
   A_3126_MXZ01MA.A_3126_MXZ01.Par.spare46 := FALSE;
   A_3126_MXZ01MA.A_3126_MXZ01.Par.OutEdgeFaultReset := FALSE;
   A_3126_MXZ01MA.A_3126_MXZ01.Par.OutDelayFault := FALSE;
   A_3126_MXZ01MA.A_3126_MXZ01.Par.OutFlagFaultDev := FALSE;
   A_3126_MXZ01MA.A_3126_MXZ01.Par.ParMonTime := 20;
   A_3126_MXZ01MA.A_3126_MXZ01.Par.ParStartingTime := 1800;
   A_3126_MXZ01MA.A_3126_MXZ01.Par.ParStoppingTime := 1200;
   A_3126_MXZ01MA.A_3126_MXZ01.Par.ParIdlingTime := 0;
   A_3126_MXZ01MA.A_3126_MXZ01.Par.ParDelayTime := 10;
   A_3126_MXZ01MA.A_3126_MXZ01.Par.OutMonTime := 0;
   A_3126_MXZ01MA.A_3126_MXZ01.Par.OutTransitionTime := 0;
   A_3126_MXZ01MA.A_3126_MXZ01.Par.OutDelayTime := 0;
   A_3126_MXZ01MA.A_3126_MXZ01.Par.InOutManPulseLen := 0;
    A_3126_TSC01_AC.StCode := 0;
   A_3126_TSC01_AC.InMonLL := FALSE;
   A_3126_TSC01_AC.InMonL := FALSE;
   A_3126_TSC01_AC.InMonMid := FALSE;
   A_3126_TSC01_AC.InMonH := FALSE;
   A_3126_TSC01_AC.InMonHH := FALSE;
   A_3126_TSC01_AC.spare0205 := FALSE;
   A_3126_TSC01_AC.InpFaultAI := FALSE;
   A_3126_TSC01_AC.InpFaultDev := FALSE;
   A_3126_TSC01_AC.InHWStop := FALSE;
   A_3126_TSC01_AC.InDPFault := FALSE;
   A_3126_TSC01_AC.InDisable := FALSE;
   A_3126_TSC01_AC.CmdFaultReset := FALSE;
   A_3126_TSC01_AC.InLocal := FALSE;
   A_3126_TSC01_AC.spare0305 := FALSE;
   A_3126_TSC01_AC.InReport := FALSE;
   A_3126_TSC01_AC.spare0307 := FALSE;
   A_3126_TSC01_AC.OutLL := FALSE;
   A_3126_TSC01_AC.OutL := FALSE;
   A_3126_TSC01_AC.OutH := FALSE;
   A_3126_TSC01_AC.OutHH := FALSE;
   A_3126_TSC01_AC.OutOverflow := FALSE;
   A_3126_TSC01_AC.spare0405 := FALSE;
   A_3126_TSC01_AC.OutFaultAI := FALSE;
   A_3126_TSC01_AC.spare0407 := FALSE;
   A_3126_TSC01_AC.StLL := FALSE;
   A_3126_TSC01_AC.StL := FALSE;
   A_3126_TSC01_AC.StMid := FALSE;
   A_3126_TSC01_AC.StH := FALSE;
   A_3126_TSC01_AC.StHH := FALSE;
   A_3126_TSC01_AC.StFaultAI := FALSE;
   A_3126_TSC01_AC.OutWarning := FALSE;
   A_3126_TSC01_AC.OutFaulted := FALSE;
   A_3126_TSC01_AC.InpValue := 0;
   A_3126_TSC01_AC.OutValuePc := 0;
   A_3126_TSC01_AC.OutValueUnits := L#0;
   A_3126_TSC01_AC.Msg.WarningDoneLL := FALSE;
   A_3126_TSC01_AC.Msg.WarningDoneL := FALSE;
   A_3126_TSC01_AC.Msg.WarningDoneMid := FALSE;
   A_3126_TSC01_AC.Msg.WarningDoneH := FALSE;
   A_3126_TSC01_AC.Msg.WarningDoneHH := FALSE;
   A_3126_TSC01_AC.Msg.FaultDoneLL := FALSE;
   A_3126_TSC01_AC.Msg.FaultDoneL := FALSE;
   A_3126_TSC01_AC.Msg.FaultDoneMid := FALSE;
   A_3126_TSC01_AC.Msg.FaultDoneH := FALSE;
   A_3126_TSC01_AC.Msg.FaultDoneHH := FALSE;
   A_3126_TSC01_AC.Msg.FaultDoneDev := FALSE;
   A_3126_TSC01_AC.Msg.FaultDoneAI := FALSE;
   A_3126_TSC01_AC.OutAlarmNrLog := 0;
   A_3126_TSC01_AC.Par.ParObjectNo := 27124;
   A_3126_TSC01_AC.Par.ParMsgType := 7252;
   A_3126_TSC01_AC.Par.ParHornCode := 10;
   A_3126_TSC01_AC.Par.ParLogOff := FALSE;
   A_3126_TSC01_AC.Par.ParSpare0401 := FALSE;
   A_3126_TSC01_AC.Par.ParValueByUser := FALSE;
   A_3126_TSC01_AC.Par.ParLimitsPc := TRUE;
   A_3126_TSC01_AC.Par.ParWago := FALSE;
   A_3126_TSC01_AC.Par.ParNoHornByWarning := FALSE;
   A_3126_TSC01_AC.Par.ParWarningLL := FALSE;
   A_3126_TSC01_AC.Par.ParWarningL := FALSE;
   A_3126_TSC01_AC.Par.ParWarningMid := FALSE;
   A_3126_TSC01_AC.Par.ParWarningH := FALSE;
   A_3126_TSC01_AC.Par.ParWarningHH := FALSE;
   A_3126_TSC01_AC.Par.ParPreAlarmLL := FALSE;
   A_3126_TSC01_AC.Par.ParPreAlarmL := FALSE;
   A_3126_TSC01_AC.Par.ParPreAlarmMid := FALSE;
   A_3126_TSC01_AC.Par.ParPreAlarmH := FALSE;
   A_3126_TSC01_AC.Par.ParPreAlarmHH := FALSE;
   A_3126_TSC01_AC.Par.ParUnitsByZeroDigit := L#0;
   A_3126_TSC01_AC.Par.ParUnitsByMaxDigit := L#25384;
   A_3126_TSC01_AC.Par.ParUnitsBy100Pc := L#10000;
   A_3126_TSC01_AC.Par.ParLimitLL := L#-1;
   A_3126_TSC01_AC.Par.ParLimitL := L#0;
   A_3126_TSC01_AC.Par.ParLimitH := L#5400;
   A_3126_TSC01_AC.Par.ParLimitHH := L#6000;
   A_3126_TSC01_AC.Par.ParMonTimeLL := 0;
   A_3126_TSC01_AC.Par.ParMonTimeL := 0;
   A_3126_TSC01_AC.Par.ParMonTimeMid := 0;
   A_3126_TSC01_AC.Par.ParMonTimeH := 0;
   A_3126_TSC01_AC.Par.ParMonTimeHH := 0;
   A_3126_TSC01_AC.Par.ParDelayTimeDown := 10;
   A_3126_TSC01_AC.Par.ParDelayTimeUp := 10;
   A_3126_TSC01_AC.Par.ParDelayTime := 30;
   A_3126_TSC01_AC.Par.OutMonTimeLL := 0;
   A_3126_TSC01_AC.Par.OutMonTimeL := 0;
   A_3126_TSC01_AC.Par.OutMonTimeMid := 0;
   A_3126_TSC01_AC.Par.OutMonTimeH := 0;
   A_3126_TSC01_AC.Par.OutMonTimeHH := 0;
   A_3126_TSC01_AC.Par.OutDelayTimeDown := 0;
   A_3126_TSC01_AC.Par.OutDelayTimeUp := 0;
   A_3126_TSC01_AC.Par.OutDelayTime := 0;
   A_3126_TSC01_AC.Par.Spare66 := 0;
   A_3126_TSC01_AF.StCode := 0;
   A_3126_TSC01_AF.InMonLL := FALSE;
   A_3126_TSC01_AF.InMonL := FALSE;
   A_3126_TSC01_AF.InMonMid := FALSE;
   A_3126_TSC01_AF.InMonH := FALSE;
   A_3126_TSC01_AF.InMonHH := FALSE;
   A_3126_TSC01_AF.spare0205 := FALSE;
   A_3126_TSC01_AF.InpFaultAI := FALSE;
   A_3126_TSC01_AF.InpFaultDev := FALSE;
   A_3126_TSC01_AF.InHWStop := FALSE;
   A_3126_TSC01_AF.InDPFault := FALSE;
   A_3126_TSC01_AF.InDisable := FALSE;
   A_3126_TSC01_AF.CmdFaultReset := FALSE;
   A_3126_TSC01_AF.InLocal := FALSE;
   A_3126_TSC01_AF.spare0305 := FALSE;
   A_3126_TSC01_AF.InReport := FALSE;
   A_3126_TSC01_AF.spare0307 := FALSE;
   A_3126_TSC01_AF.OutLL := FALSE;
   A_3126_TSC01_AF.OutL := FALSE;
   A_3126_TSC01_AF.OutH := FALSE;
   A_3126_TSC01_AF.OutHH := FALSE;
   A_3126_TSC01_AF.OutOverflow := FALSE;
   A_3126_TSC01_AF.spare0405 := FALSE;
   A_3126_TSC01_AF.OutFaultAI := FALSE;
   A_3126_TSC01_AF.spare0407 := FALSE;
   A_3126_TSC01_AF.StLL := FALSE;
   A_3126_TSC01_AF.StL := FALSE;
   A_3126_TSC01_AF.StMid := FALSE;
   A_3126_TSC01_AF.StH := FALSE;
   A_3126_TSC01_AF.StHH := FALSE;
   A_3126_TSC01_AF.StFaultAI := FALSE;
   A_3126_TSC01_AF.OutWarning := FALSE;
   A_3126_TSC01_AF.OutFaulted := FALSE;
   A_3126_TSC01_AF.InpValue := 0;
   A_3126_TSC01_AF.OutValuePc := 0;
   A_3126_TSC01_AF.OutValueUnits := L#0;
   A_3126_TSC01_AF.Msg.WarningDoneLL := FALSE;
   A_3126_TSC01_AF.Msg.WarningDoneL := FALSE;
   A_3126_TSC01_AF.Msg.WarningDoneMid := FALSE;
   A_3126_TSC01_AF.Msg.WarningDoneH := FALSE;
   A_3126_TSC01_AF.Msg.WarningDoneHH := FALSE;
   A_3126_TSC01_AF.Msg.FaultDoneLL := FALSE;
   A_3126_TSC01_AF.Msg.FaultDoneL := FALSE;
   A_3126_TSC01_AF.Msg.FaultDoneMid := FALSE;
   A_3126_TSC01_AF.Msg.FaultDoneH := FALSE;
   A_3126_TSC01_AF.Msg.FaultDoneHH := FALSE;
   A_3126_TSC01_AF.Msg.FaultDoneDev := FALSE;
   A_3126_TSC01_AF.Msg.FaultDoneAI := FALSE;
   A_3126_TSC01_AF.OutAlarmNrLog := 0;
   A_3126_TSC01_AF.Par.ParObjectNo := 27125;
   A_3126_TSC01_AF.Par.ParMsgType := 7252;
   A_3126_TSC01_AF.Par.ParHornCode := 10;
   A_3126_TSC01_AF.Par.ParLogOff := FALSE;
   A_3126_TSC01_AF.Par.ParSpare0401 := FALSE;
   A_3126_TSC01_AF.Par.ParValueByUser := FALSE;
   A_3126_TSC01_AF.Par.ParLimitsPc := TRUE;
   A_3126_TSC01_AF.Par.ParWago := FALSE;
   A_3126_TSC01_AF.Par.ParNoHornByWarning := FALSE;
   A_3126_TSC01_AF.Par.ParWarningLL := FALSE;
   A_3126_TSC01_AF.Par.ParWarningL := FALSE;
   A_3126_TSC01_AF.Par.ParWarningMid := FALSE;
   A_3126_TSC01_AF.Par.ParWarningH := FALSE;
   A_3126_TSC01_AF.Par.ParWarningHH := FALSE;
   A_3126_TSC01_AF.Par.ParPreAlarmLL := FALSE;
   A_3126_TSC01_AF.Par.ParPreAlarmL := FALSE;
   A_3126_TSC01_AF.Par.ParPreAlarmMid := FALSE;
   A_3126_TSC01_AF.Par.ParPreAlarmH := FALSE;
   A_3126_TSC01_AF.Par.ParPreAlarmHH := FALSE;
   A_3126_TSC01_AF.Par.ParUnitsByZeroDigit := L#0;
   A_3126_TSC01_AF.Par.ParUnitsByMaxDigit := L#16880;
   A_3126_TSC01_AF.Par.ParUnitsBy100Pc := L#10000;
   A_3126_TSC01_AF.Par.ParLimitLL := L#-1;
   A_3126_TSC01_AF.Par.ParLimitL := L#3000;
   A_3126_TSC01_AF.Par.ParLimitH := L#10000;
   A_3126_TSC01_AF.Par.ParLimitHH := L#10100;
   A_3126_TSC01_AF.Par.ParMonTimeLL := 0;
   A_3126_TSC01_AF.Par.ParMonTimeL := 0;
   A_3126_TSC01_AF.Par.ParMonTimeMid := 0;
   A_3126_TSC01_AF.Par.ParMonTimeH := 0;
   A_3126_TSC01_AF.Par.ParMonTimeHH := 0;
   A_3126_TSC01_AF.Par.ParDelayTimeDown := 10;
   A_3126_TSC01_AF.Par.ParDelayTimeUp := 10;
   A_3126_TSC01_AF.Par.ParDelayTime := 30;
   A_3126_TSC01_AF.Par.OutMonTimeLL := 0;
   A_3126_TSC01_AF.Par.OutMonTimeL := 0;
   A_3126_TSC01_AF.Par.OutMonTimeMid := 0;
   A_3126_TSC01_AF.Par.OutMonTimeH := 0;
   A_3126_TSC01_AF.Par.OutMonTimeHH := 0;
   A_3126_TSC01_AF.Par.OutDelayTimeDown := 0;
   A_3126_TSC01_AF.Par.OutDelayTimeUp := 0;
   A_3126_TSC01_AF.Par.OutDelayTime := 0;
   A_3126_TSC01_AF.Par.Spare66 := 0;
   A_3126_TSC01_AP.StCode := 0;
   A_3126_TSC01_AP.InMonLL := FALSE;
   A_3126_TSC01_AP.InMonL := FALSE;
   A_3126_TSC01_AP.InMonMid := FALSE;
   A_3126_TSC01_AP.InMonH := FALSE;
   A_3126_TSC01_AP.InMonHH := FALSE;
   A_3126_TSC01_AP.spare0205 := FALSE;
   A_3126_TSC01_AP.InpFaultAI := FALSE;
   A_3126_TSC01_AP.InpFaultDev := FALSE;
   A_3126_TSC01_AP.InHWStop := FALSE;
   A_3126_TSC01_AP.InDPFault := FALSE;
   A_3126_TSC01_AP.InDisable := FALSE;
   A_3126_TSC01_AP.CmdFaultReset := FALSE;
   A_3126_TSC01_AP.InLocal := FALSE;
   A_3126_TSC01_AP.spare0305 := FALSE;
   A_3126_TSC01_AP.InReport := FALSE;
   A_3126_TSC01_AP.spare0307 := FALSE;
   A_3126_TSC01_AP.OutLL := FALSE;
   A_3126_TSC01_AP.OutL := FALSE;
   A_3126_TSC01_AP.OutH := FALSE;
   A_3126_TSC01_AP.OutHH := FALSE;
   A_3126_TSC01_AP.OutOverflow := FALSE;
   A_3126_TSC01_AP.spare0405 := FALSE;
   A_3126_TSC01_AP.OutFaultAI := FALSE;
   A_3126_TSC01_AP.spare0407 := FALSE;
   A_3126_TSC01_AP.StLL := FALSE;
   A_3126_TSC01_AP.StL := FALSE;
   A_3126_TSC01_AP.StMid := FALSE;
   A_3126_TSC01_AP.StH := FALSE;
   A_3126_TSC01_AP.StHH := FALSE;
   A_3126_TSC01_AP.StFaultAI := FALSE;
   A_3126_TSC01_AP.OutWarning := FALSE;
   A_3126_TSC01_AP.OutFaulted := FALSE;
   A_3126_TSC01_AP.InpValue := 0;
   A_3126_TSC01_AP.OutValuePc := 0;
   A_3126_TSC01_AP.OutValueUnits := L#0;
   A_3126_TSC01_AP.Msg.WarningDoneLL := FALSE;
   A_3126_TSC01_AP.Msg.WarningDoneL := FALSE;
   A_3126_TSC01_AP.Msg.WarningDoneMid := FALSE;
   A_3126_TSC01_AP.Msg.WarningDoneH := FALSE;
   A_3126_TSC01_AP.Msg.WarningDoneHH := FALSE;
   A_3126_TSC01_AP.Msg.FaultDoneLL := FALSE;
   A_3126_TSC01_AP.Msg.FaultDoneL := FALSE;
   A_3126_TSC01_AP.Msg.FaultDoneMid := FALSE;
   A_3126_TSC01_AP.Msg.FaultDoneH := FALSE;
   A_3126_TSC01_AP.Msg.FaultDoneHH := FALSE;
   A_3126_TSC01_AP.Msg.FaultDoneDev := FALSE;
   A_3126_TSC01_AP.Msg.FaultDoneAI := FALSE;
   A_3126_TSC01_AP.OutAlarmNrLog := 0;
   A_3126_TSC01_AP.Par.ParObjectNo := 27126;
   A_3126_TSC01_AP.Par.ParMsgType := 7252;
   A_3126_TSC01_AP.Par.ParHornCode := 10;
   A_3126_TSC01_AP.Par.ParLogOff := FALSE;
   A_3126_TSC01_AP.Par.ParSpare0401 := FALSE;
   A_3126_TSC01_AP.Par.ParValueByUser := FALSE;
   A_3126_TSC01_AP.Par.ParLimitsPc := TRUE;
   A_3126_TSC01_AP.Par.ParWago := FALSE;
   A_3126_TSC01_AP.Par.ParNoHornByWarning := FALSE;
   A_3126_TSC01_AP.Par.ParWarningLL := FALSE;
   A_3126_TSC01_AP.Par.ParWarningL := FALSE;
   A_3126_TSC01_AP.Par.ParWarningMid := FALSE;
   A_3126_TSC01_AP.Par.ParWarningH := FALSE;
   A_3126_TSC01_AP.Par.ParWarningHH := FALSE;
   A_3126_TSC01_AP.Par.ParPreAlarmLL := FALSE;
   A_3126_TSC01_AP.Par.ParPreAlarmL := FALSE;
   A_3126_TSC01_AP.Par.ParPreAlarmMid := FALSE;
   A_3126_TSC01_AP.Par.ParPreAlarmH := FALSE;
   A_3126_TSC01_AP.Par.ParPreAlarmHH := FALSE;
   A_3126_TSC01_AP.Par.ParUnitsByZeroDigit := L#0;
   A_3126_TSC01_AP.Par.ParUnitsByMaxDigit := L#16384;
   A_3126_TSC01_AP.Par.ParUnitsBy100Pc := L#10000;
   A_3126_TSC01_AP.Par.ParLimitLL := L#-1;
   A_3126_TSC01_AP.Par.ParLimitL := L#0;
   A_3126_TSC01_AP.Par.ParLimitH := L#3150;
   A_3126_TSC01_AP.Par.ParLimitHH := L#3500;
   A_3126_TSC01_AP.Par.ParMonTimeLL := 0;
   A_3126_TSC01_AP.Par.ParMonTimeL := 0;
   A_3126_TSC01_AP.Par.ParMonTimeMid := 0;
   A_3126_TSC01_AP.Par.ParMonTimeH := 0;
   A_3126_TSC01_AP.Par.ParMonTimeHH := 0;
   A_3126_TSC01_AP.Par.ParDelayTimeDown := 10;
   A_3126_TSC01_AP.Par.ParDelayTimeUp := 10;
   A_3126_TSC01_AP.Par.ParDelayTime := 30;
   A_3126_TSC01_AP.Par.OutMonTimeLL := 0;
   A_3126_TSC01_AP.Par.OutMonTimeL := 0;
   A_3126_TSC01_AP.Par.OutMonTimeMid := 0;
   A_3126_TSC01_AP.Par.OutMonTimeH := 0;
   A_3126_TSC01_AP.Par.OutMonTimeHH := 0;
   A_3126_TSC01_AP.Par.OutDelayTimeDown := 0;
   A_3126_TSC01_AP.Par.OutDelayTimeUp := 0;
   A_3126_TSC01_AP.Par.OutDelayTime := 0;
   A_3126_TSC01_AP.Par.Spare66 := 0;
   A_3126_TSC01_AT.StCode := 0;
   A_3126_TSC01_AT.InMonLL := FALSE;
   A_3126_TSC01_AT.InMonL := FALSE;
   A_3126_TSC01_AT.InMonMid := FALSE;
   A_3126_TSC01_AT.InMonH := FALSE;
   A_3126_TSC01_AT.InMonHH := FALSE;
   A_3126_TSC01_AT.spare0205 := FALSE;
   A_3126_TSC01_AT.InpFaultAI := FALSE;
   A_3126_TSC01_AT.InpFaultDev := FALSE;
   A_3126_TSC01_AT.InHWStop := FALSE;
   A_3126_TSC01_AT.InDPFault := FALSE;
   A_3126_TSC01_AT.InDisable := FALSE;
   A_3126_TSC01_AT.CmdFaultReset := FALSE;
   A_3126_TSC01_AT.InLocal := FALSE;
   A_3126_TSC01_AT.spare0305 := FALSE;
   A_3126_TSC01_AT.InReport := FALSE;
   A_3126_TSC01_AT.spare0307 := FALSE;
   A_3126_TSC01_AT.OutLL := FALSE;
   A_3126_TSC01_AT.OutL := FALSE;
   A_3126_TSC01_AT.OutH := FALSE;
   A_3126_TSC01_AT.OutHH := FALSE;
   A_3126_TSC01_AT.OutOverflow := FALSE;
   A_3126_TSC01_AT.spare0405 := FALSE;
   A_3126_TSC01_AT.OutFaultAI := FALSE;
   A_3126_TSC01_AT.spare0407 := FALSE;
   A_3126_TSC01_AT.StLL := FALSE;
   A_3126_TSC01_AT.StL := FALSE;
   A_3126_TSC01_AT.StMid := FALSE;
   A_3126_TSC01_AT.StH := FALSE;
   A_3126_TSC01_AT.StHH := FALSE;
   A_3126_TSC01_AT.StFaultAI := FALSE;
   A_3126_TSC01_AT.OutWarning := FALSE;
   A_3126_TSC01_AT.OutFaulted := FALSE;
   A_3126_TSC01_AT.InpValue := 0;
   A_3126_TSC01_AT.OutValuePc := 0;
   A_3126_TSC01_AT.OutValueUnits := L#0;
   A_3126_TSC01_AT.Msg.WarningDoneLL := FALSE;
   A_3126_TSC01_AT.Msg.WarningDoneL := FALSE;
   A_3126_TSC01_AT.Msg.WarningDoneMid := FALSE;
   A_3126_TSC01_AT.Msg.WarningDoneH := FALSE;
   A_3126_TSC01_AT.Msg.WarningDoneHH := FALSE;
   A_3126_TSC01_AT.Msg.FaultDoneLL := FALSE;
   A_3126_TSC01_AT.Msg.FaultDoneL := FALSE;
   A_3126_TSC01_AT.Msg.FaultDoneMid := FALSE;
   A_3126_TSC01_AT.Msg.FaultDoneH := FALSE;
   A_3126_TSC01_AT.Msg.FaultDoneHH := FALSE;
   A_3126_TSC01_AT.Msg.FaultDoneDev := FALSE;
   A_3126_TSC01_AT.Msg.FaultDoneAI := FALSE;
   A_3126_TSC01_AT.OutAlarmNrLog := 0;
   A_3126_TSC01_AT.Par.ParObjectNo := 27127;
   A_3126_TSC01_AT.Par.ParMsgType := 7252;
   A_3126_TSC01_AT.Par.ParHornCode := 10;
   A_3126_TSC01_AT.Par.ParLogOff := FALSE;
   A_3126_TSC01_AT.Par.ParSpare0401 := FALSE;
   A_3126_TSC01_AT.Par.ParValueByUser := FALSE;
   A_3126_TSC01_AT.Par.ParLimitsPc := TRUE;
   A_3126_TSC01_AT.Par.ParWago := FALSE;
   A_3126_TSC01_AT.Par.ParNoHornByWarning := FALSE;
   A_3126_TSC01_AT.Par.ParWarningLL := FALSE;
   A_3126_TSC01_AT.Par.ParWarningL := FALSE;
   A_3126_TSC01_AT.Par.ParWarningMid := FALSE;
   A_3126_TSC01_AT.Par.ParWarningH := FALSE;
   A_3126_TSC01_AT.Par.ParWarningHH := FALSE;
   A_3126_TSC01_AT.Par.ParPreAlarmLL := FALSE;
   A_3126_TSC01_AT.Par.ParPreAlarmL := FALSE;
   A_3126_TSC01_AT.Par.ParPreAlarmMid := FALSE;
   A_3126_TSC01_AT.Par.ParPreAlarmH := FALSE;
   A_3126_TSC01_AT.Par.ParPreAlarmHH := FALSE;
   A_3126_TSC01_AT.Par.ParUnitsByZeroDigit := L#0;
   A_3126_TSC01_AT.Par.ParUnitsByMaxDigit := L#16384;
   A_3126_TSC01_AT.Par.ParUnitsBy100Pc := L#10000;
   A_3126_TSC01_AT.Par.ParLimitLL := L#-1;
   A_3126_TSC01_AT.Par.ParLimitL := L#0;
   A_3126_TSC01_AT.Par.ParLimitH := L#7000;
   A_3126_TSC01_AT.Par.ParLimitHH := L#8000;
   A_3126_TSC01_AT.Par.ParMonTimeLL := 0;
   A_3126_TSC01_AT.Par.ParMonTimeL := 0;
   A_3126_TSC01_AT.Par.ParMonTimeMid := 0;
   A_3126_TSC01_AT.Par.ParMonTimeH := 0;
   A_3126_TSC01_AT.Par.ParMonTimeHH := 0;
   A_3126_TSC01_AT.Par.ParDelayTimeDown := 10;
   A_3126_TSC01_AT.Par.ParDelayTimeUp := 10;
   A_3126_TSC01_AT.Par.ParDelayTime := 30;
   A_3126_TSC01_AT.Par.OutMonTimeLL := 0;
   A_3126_TSC01_AT.Par.OutMonTimeL := 0;
   A_3126_TSC01_AT.Par.OutMonTimeMid := 0;
   A_3126_TSC01_AT.Par.OutMonTimeH := 0;
   A_3126_TSC01_AT.Par.OutMonTimeHH := 0;
   A_3126_TSC01_AT.Par.OutDelayTimeDown := 0;
   A_3126_TSC01_AT.Par.OutDelayTimeUp := 0;
   A_3126_TSC01_AT.Par.OutDelayTime := 0;
   A_3126_TSC01_AT.Par.Spare66 := 0;
   A_3125_TSC01.StCode := 0;
   A_3125_TSC01.InMonTrue := FALSE;
   A_3125_TSC01.InMonFalse := FALSE;
   A_3125_TSC01.InPreAlarmTrue := FALSE;
   A_3125_TSC01.InPreAlarmFalse := FALSE;
   A_3125_TSC01.InStopTrueTime := FALSE;
   A_3125_TSC01.InStopFalseTime := FALSE;
   A_3125_TSC01.InpTrue := FALSE;
   A_3125_TSC01.InpFaultDev := FALSE;
   A_3125_TSC01.CmdRstTrueTime := FALSE;
   A_3125_TSC01.CmdRstFalseTime := FALSE;
   A_3125_TSC01.CmdRunTimeoutTime := FALSE;
   A_3125_TSC01.CmdFaultReset := FALSE;
   A_3125_TSC01.InLocal := FALSE;
   A_3125_TSC01.spare0305 := FALSE;
   A_3125_TSC01.InReport := FALSE;
   A_3125_TSC01.OutTimeoutTime := FALSE;
   A_3125_TSC01.InHWStop := FALSE;
   A_3125_TSC01.InDPFault := FALSE;
   A_3125_TSC01.OutPreAlarmTrue := FALSE;
   A_3125_TSC01.OutPreAlarmFalse := FALSE;
   A_3125_TSC01.OutFlagPos := FALSE;
   A_3125_TSC01.OutFlagNeg := FALSE;
   A_3125_TSC01.OutpFaultReset := FALSE;
   A_3125_TSC01.OutTrue := FALSE;
   A_3125_TSC01.StFalse := FALSE;
   A_3125_TSC01.StCtoTrue := FALSE;
   A_3125_TSC01.StTrue := FALSE;
   A_3125_TSC01.StCtoFalse := FALSE;
   A_3125_TSC01.StFault := FALSE;
   A_3125_TSC01.OutAlarmNrLog := 0;
   A_3125_TSC01.Par.ParObjectNo := 27107;
   A_3125_TSC01.Par.ParMsgType := 7156;
   A_3125_TSC01.Par.ParHornCode := 0;
   A_3125_TSC01.Par.ParLogOff := FALSE;
   A_3125_TSC01.Par.spare0401 := FALSE;
   A_3125_TSC01.Par.Par2WorkingCond := FALSE;
   A_3125_TSC01.Par.ParFaultRetry := FALSE;
   A_3125_TSC01.Par.ParBinLevel := FALSE;
   A_3125_TSC01.Par.ParDelayChange := 20;
   A_3125_TSC01.Par.ParDelayTrue := 10;
   A_3125_TSC01.Par.ParDelayFalse := 0;
   A_3125_TSC01.Par.ParTimeoutTrue := 0;
   A_3125_TSC01.Par.ParTimeoutFalse := 0;
   A_3125_TSC01.Par.OutMonTime := 0;
   A_3125_TSC01.Par.OutTransitionTime := 0;
   A_3125_TSC01.Par.OutMonTrue := FALSE;
   A_3125_TSC01.Par.OutMonFalse := FALSE;
   A_3125_TSC01.Par.OutFlagFaultDev := FALSE;
   A_3125_TSC01.Par.OutDelayTime := 0;
   A_3126_TSC01.StCode := 0;
   A_3126_TSC01.InMonTrue := FALSE;
   A_3126_TSC01.InMonFalse := FALSE;
   A_3126_TSC01.InPreAlarmTrue := FALSE;
   A_3126_TSC01.InPreAlarmFalse := FALSE;
   A_3126_TSC01.InStopTrueTime := FALSE;
   A_3126_TSC01.InStopFalseTime := FALSE;
   A_3126_TSC01.InpTrue := FALSE;
   A_3126_TSC01.InpFaultDev := FALSE;
   A_3126_TSC01.CmdRstTrueTime := FALSE;
   A_3126_TSC01.CmdRstFalseTime := FALSE;
   A_3126_TSC01.CmdRunTimeoutTime := FALSE;
   A_3126_TSC01.CmdFaultReset := FALSE;
   A_3126_TSC01.InLocal := FALSE;
   A_3126_TSC01.spare0305 := FALSE;
   A_3126_TSC01.InReport := FALSE;
   A_3126_TSC01.OutTimeoutTime := FALSE;
   A_3126_TSC01.InHWStop := FALSE;
   A_3126_TSC01.InDPFault := FALSE;
   A_3126_TSC01.OutPreAlarmTrue := FALSE;
   A_3126_TSC01.OutPreAlarmFalse := FALSE;
   A_3126_TSC01.OutFlagPos := FALSE;
   A_3126_TSC01.OutFlagNeg := FALSE;
   A_3126_TSC01.OutpFaultReset := FALSE;
   A_3126_TSC01.OutTrue := FALSE;
   A_3126_TSC01.StFalse := FALSE;
   A_3126_TSC01.StCtoTrue := FALSE;
   A_3126_TSC01.StTrue := FALSE;
   A_3126_TSC01.StCtoFalse := FALSE;
   A_3126_TSC01.StFault := FALSE;
   A_3126_TSC01.OutAlarmNrLog := 0;
   A_3126_TSC01.Par.ParObjectNo := 27128;
   A_3126_TSC01.Par.ParMsgType := 7156;
   A_3126_TSC01.Par.ParHornCode := 0;
   A_3126_TSC01.Par.ParLogOff := FALSE;
   A_3126_TSC01.Par.spare0401 := FALSE;
   A_3126_TSC01.Par.Par2WorkingCond := FALSE;
   A_3126_TSC01.Par.ParFaultRetry := FALSE;
   A_3126_TSC01.Par.ParBinLevel := FALSE;
   A_3126_TSC01.Par.ParDelayChange := 20;
   A_3126_TSC01.Par.ParDelayTrue := 10;
   A_3126_TSC01.Par.ParDelayFalse := 0;
   A_3126_TSC01.Par.ParTimeoutTrue := 0;
   A_3126_TSC01.Par.ParTimeoutFalse := 0;
   A_3126_TSC01.Par.OutMonTime := 0;
   A_3126_TSC01.Par.OutTransitionTime := 0;
   A_3126_TSC01.Par.OutMonTrue := FALSE;
   A_3126_TSC01.Par.OutMonFalse := FALSE;
   A_3126_TSC01.Par.OutFlagFaultDev := FALSE;
   A_3126_TSC01.Par.OutDelayTime := 0;
   A_3125_MXZ02MA.Ma.StCode := 0;
   A_3125_MXZ02MA.Ma.InEnableRev := FALSE;
   A_3125_MXZ02MA.Ma.InEnableFwd := FALSE;
   A_3125_MXZ02MA.Ma.InOverrideHLOutlet := FALSE;
   A_3125_MXZ02MA.Ma.spare0203 := FALSE;
   A_3125_MXZ02MA.Ma.OutEdgeFaultReset := FALSE;
   A_3125_MXZ02MA.Ma.OutFaultResetFcttst := FALSE;
   A_3125_MXZ02MA.Ma.InpControlEBM := FALSE;
   A_3125_MXZ02MA.Ma.InpLocked := FALSE;
   A_3125_MXZ02MA.Ma.CmdOff := FALSE;
   A_3125_MXZ02MA.Ma.CmdOn := FALSE;
   A_3125_MXZ02MA.Ma.CmdNext := FALSE;
   A_3125_MXZ02MA.Ma.CmdFaultReset := FALSE;
   A_3125_MXZ02MA.Ma.InLocal := FALSE;
   A_3125_MXZ02MA.Ma.InManual := FALSE;
   A_3125_MXZ02MA.Ma.CmdTestEBM := FALSE;
   A_3125_MXZ02MA.Ma.InSeqStop := FALSE;
   A_3125_MXZ02MA.Ma.OutWarning := FALSE;
   A_3125_MXZ02MA.Ma.InfBMTopOk := FALSE;
   A_3125_MXZ02MA.Ma.InfBMBottomOk := FALSE;
   A_3125_MXZ02MA.Ma.InfSMOk := FALSE;
   A_3125_MXZ02MA.Ma.OutpFcttst_BM_Top := FALSE;
   A_3125_MXZ02MA.Ma.OutpFcttst_BM_Bottom := FALSE;
   A_3125_MXZ02MA.Ma.OutpFcttst_SM := FALSE;
   A_3125_MXZ02MA.Ma.OutpFaultReset := FALSE;
   A_3125_MXZ02MA.Ma.StStopped := FALSE;
   A_3125_MXZ02MA.Ma.StStarting := FALSE;
   A_3125_MXZ02MA.Ma.StStartedFwd := FALSE;
   A_3125_MXZ02MA.Ma.StStopping := FALSE;
   A_3125_MXZ02MA.Ma.StFault := FALSE;
   A_3125_MXZ02MA.Ma.StStartedRev := FALSE;
   A_3125_MXZ02MA.Ma.StLocked := FALSE;
   A_3125_MXZ02MA.Ma.OutTestTime := 0;
   A_3125_MXZ02MA.Ma.Par.ParObjectNo := 27108;
   A_3125_MXZ02MA.Ma.Par.ParWithMon1 := TRUE;
   A_3125_MXZ02MA.Ma.Par.ParWithMon3 := FALSE;
   A_3125_MXZ02MA.Ma.Par.ParWithMon4 := FALSE;
   A_3125_MXZ02MA.Ma.Par.ParWithMon5 := FALSE;
   A_3125_MXZ02MA.Ma.Par.ParWithMon6 := FALSE;
   A_3125_MXZ02MA.Ma.Par.ParMon1IsHL := FALSE;
   A_3125_MXZ02MA.Ma.Par.ParMon1IsLS := TRUE;
   A_3125_MXZ02MA.Ma.Par.ParMon1StopByFault := TRUE;
   A_3125_MXZ02MA.Ma.Par.ParMon2IsLS := FALSE;
   A_3125_MXZ02MA.Ma.Par.ParMon3IsLS := FALSE;
   A_3125_MXZ02MA.Ma.Par.ParMon4AsWarning := FALSE;
   A_3125_MXZ02MA.Ma.Par.ParMon4StopByFault := FALSE;
   A_3125_MXZ02MA.Ma.Par.ParMon4IsLS := FALSE;
   A_3125_MXZ02MA.Ma.Par.ParEBM := FALSE;
   A_3125_MXZ02MA.Ma.Par.ParMon4IsSM := FALSE;
   A_3125_MXZ02MA.A_3125_BFT09.StCode := 0;
   A_3125_MXZ02MA.A_3125_BFT09.InMonTrue := FALSE;
   A_3125_MXZ02MA.A_3125_BFT09.InMonFalse := FALSE;
   A_3125_MXZ02MA.A_3125_BFT09.InPreAlarmTrue := FALSE;
   A_3125_MXZ02MA.A_3125_BFT09.InPreAlarmFalse := FALSE;
   A_3125_MXZ02MA.A_3125_BFT09.InStopTrueTime := FALSE;
   A_3125_MXZ02MA.A_3125_BFT09.InStopFalseTime := FALSE;
   A_3125_MXZ02MA.A_3125_BFT09.InpTrue := FALSE;
   A_3125_MXZ02MA.A_3125_BFT09.InpFaultDev := FALSE;
   A_3125_MXZ02MA.A_3125_BFT09.CmdRstTrueTime := FALSE;
   A_3125_MXZ02MA.A_3125_BFT09.CmdRstFalseTime := FALSE;
   A_3125_MXZ02MA.A_3125_BFT09.CmdRunTimeoutTime := FALSE;
   A_3125_MXZ02MA.A_3125_BFT09.CmdFaultReset := FALSE;
   A_3125_MXZ02MA.A_3125_BFT09.InLocal := FALSE;
   A_3125_MXZ02MA.A_3125_BFT09.spare0305 := FALSE;
   A_3125_MXZ02MA.A_3125_BFT09.InReport := FALSE;
   A_3125_MXZ02MA.A_3125_BFT09.OutTimeoutTime := FALSE;
   A_3125_MXZ02MA.A_3125_BFT09.InHWStop := FALSE;
   A_3125_MXZ02MA.A_3125_BFT09.InDPFault := FALSE;
   A_3125_MXZ02MA.A_3125_BFT09.OutPreAlarmTrue := FALSE;
   A_3125_MXZ02MA.A_3125_BFT09.OutPreAlarmFalse := FALSE;
   A_3125_MXZ02MA.A_3125_BFT09.OutFlagPos := FALSE;
   A_3125_MXZ02MA.A_3125_BFT09.OutFlagNeg := FALSE;
   A_3125_MXZ02MA.A_3125_BFT09.OutpFaultReset := FALSE;
   A_3125_MXZ02MA.A_3125_BFT09.OutTrue := FALSE;
   A_3125_MXZ02MA.A_3125_BFT09.StFalse := FALSE;
   A_3125_MXZ02MA.A_3125_BFT09.StCtoTrue := FALSE;
   A_3125_MXZ02MA.A_3125_BFT09.StTrue := FALSE;
   A_3125_MXZ02MA.A_3125_BFT09.StCtoFalse := FALSE;
   A_3125_MXZ02MA.A_3125_BFT09.StFault := FALSE;
   A_3125_MXZ02MA.A_3125_BFT09.OutAlarmNrLog := 0;
   A_3125_MXZ02MA.A_3125_BFT09.Par.ParObjectNo := 27121;
   A_3125_MXZ02MA.A_3125_BFT09.Par.ParMsgType := 7135;
   A_3125_MXZ02MA.A_3125_BFT09.Par.ParHornCode := 0;
   A_3125_MXZ02MA.A_3125_BFT09.Par.ParLogOff := FALSE;
   A_3125_MXZ02MA.A_3125_BFT09.Par.spare0401 := FALSE;
   A_3125_MXZ02MA.A_3125_BFT09.Par.Par2WorkingCond := FALSE;
   A_3125_MXZ02MA.A_3125_BFT09.Par.ParFaultRetry := FALSE;
   A_3125_MXZ02MA.A_3125_BFT09.Par.ParBinLevel := FALSE;
   A_3125_MXZ02MA.A_3125_BFT09.Par.ParDelayChange := 0;
   A_3125_MXZ02MA.A_3125_BFT09.Par.ParDelayTrue := 10;
   A_3125_MXZ02MA.A_3125_BFT09.Par.ParDelayFalse := 0;
   A_3125_MXZ02MA.A_3125_BFT09.Par.ParTimeoutTrue := 0;
   A_3125_MXZ02MA.A_3125_BFT09.Par.ParTimeoutFalse := 0;
   A_3125_MXZ02MA.A_3125_BFT09.Par.OutMonTime := 0;
   A_3125_MXZ02MA.A_3125_BFT09.Par.OutTransitionTime := 0;
   A_3125_MXZ02MA.A_3125_BFT09.Par.OutMonTrue := FALSE;
   A_3125_MXZ02MA.A_3125_BFT09.Par.OutMonFalse := FALSE;
   A_3125_MXZ02MA.A_3125_BFT09.Par.OutFlagFaultDev := FALSE;
   A_3125_MXZ02MA.A_3125_BFT09.Par.OutDelayTime := 0;
   A_3125_MXZ02MA.Mon2.StCode := 0;
   A_3125_MXZ02MA.Mon2.InMonTrue := FALSE;
   A_3125_MXZ02MA.Mon2.InMonFalse := FALSE;
   A_3125_MXZ02MA.Mon2.InPreAlarmTrue := FALSE;
   A_3125_MXZ02MA.Mon2.InPreAlarmFalse := FALSE;
   A_3125_MXZ02MA.Mon2.InStopTrueTime := FALSE;
   A_3125_MXZ02MA.Mon2.InStopFalseTime := FALSE;
   A_3125_MXZ02MA.Mon2.InpTrue := FALSE;
   A_3125_MXZ02MA.Mon2.InpFaultDev := FALSE;
   A_3125_MXZ02MA.Mon2.CmdRstTrueTime := FALSE;
   A_3125_MXZ02MA.Mon2.CmdRstFalseTime := FALSE;
   A_3125_MXZ02MA.Mon2.CmdRunTimeoutTime := FALSE;
   A_3125_MXZ02MA.Mon2.CmdFaultReset := FALSE;
   A_3125_MXZ02MA.Mon2.InLocal := FALSE;
   A_3125_MXZ02MA.Mon2.spare0305 := FALSE;
   A_3125_MXZ02MA.Mon2.InReport := FALSE;
   A_3125_MXZ02MA.Mon2.OutTimeoutTime := FALSE;
   A_3125_MXZ02MA.Mon2.InHWStop := FALSE;
   A_3125_MXZ02MA.Mon2.InDPFault := FALSE;
   A_3125_MXZ02MA.Mon2.OutPreAlarmTrue := FALSE;
   A_3125_MXZ02MA.Mon2.OutPreAlarmFalse := FALSE;
   A_3125_MXZ02MA.Mon2.OutFlagPos := FALSE;
   A_3125_MXZ02MA.Mon2.OutFlagNeg := FALSE;
   A_3125_MXZ02MA.Mon2.OutpFaultReset := FALSE;
   A_3125_MXZ02MA.Mon2.OutTrue := FALSE;
   A_3125_MXZ02MA.Mon2.StFalse := FALSE;
   A_3125_MXZ02MA.Mon2.StCtoTrue := FALSE;
   A_3125_MXZ02MA.Mon2.StTrue := FALSE;
   A_3125_MXZ02MA.Mon2.StCtoFalse := FALSE;
   A_3125_MXZ02MA.Mon2.StFault := FALSE;
   A_3125_MXZ02MA.Mon2.OutAlarmNrLog := 0;
   A_3125_MXZ02MA.Mon2.Par.ParObjectNo := 0;
   A_3125_MXZ02MA.Mon2.Par.ParMsgType := 0;
   A_3125_MXZ02MA.Mon2.Par.ParHornCode := 0;
   A_3125_MXZ02MA.Mon2.Par.ParLogOff := FALSE;
   A_3125_MXZ02MA.Mon2.Par.spare0401 := FALSE;
   A_3125_MXZ02MA.Mon2.Par.Par2WorkingCond := FALSE;
   A_3125_MXZ02MA.Mon2.Par.ParFaultRetry := FALSE;
   A_3125_MXZ02MA.Mon2.Par.ParBinLevel := FALSE;
   A_3125_MXZ02MA.Mon2.Par.ParDelayChange := 0;
   A_3125_MXZ02MA.Mon2.Par.ParDelayTrue := 0;
   A_3125_MXZ02MA.Mon2.Par.ParDelayFalse := 0;
   A_3125_MXZ02MA.Mon2.Par.ParTimeoutTrue := 0;
   A_3125_MXZ02MA.Mon2.Par.ParTimeoutFalse := 0;
   A_3125_MXZ02MA.Mon2.Par.OutMonTime := 0;
   A_3125_MXZ02MA.Mon2.Par.OutTransitionTime := 0;
   A_3125_MXZ02MA.Mon2.Par.OutMonTrue := FALSE;
   A_3125_MXZ02MA.Mon2.Par.OutMonFalse := FALSE;
   A_3125_MXZ02MA.Mon2.Par.OutFlagFaultDev := FALSE;
   A_3125_MXZ02MA.Mon2.Par.OutDelayTime := 0;
   A_3125_MXZ02MA.Mon3.StCode := 0;
   A_3125_MXZ02MA.Mon3.InMonTrue := FALSE;
   A_3125_MXZ02MA.Mon3.InMonFalse := FALSE;
   A_3125_MXZ02MA.Mon3.InPreAlarmTrue := FALSE;
   A_3125_MXZ02MA.Mon3.InPreAlarmFalse := FALSE;
   A_3125_MXZ02MA.Mon3.InStopTrueTime := FALSE;
   A_3125_MXZ02MA.Mon3.InStopFalseTime := FALSE;
   A_3125_MXZ02MA.Mon3.InpTrue := FALSE;
   A_3125_MXZ02MA.Mon3.InpFaultDev := FALSE;
   A_3125_MXZ02MA.Mon3.CmdRstTrueTime := FALSE;
   A_3125_MXZ02MA.Mon3.CmdRstFalseTime := FALSE;
   A_3125_MXZ02MA.Mon3.CmdRunTimeoutTime := FALSE;
   A_3125_MXZ02MA.Mon3.CmdFaultReset := FALSE;
   A_3125_MXZ02MA.Mon3.InLocal := FALSE;
   A_3125_MXZ02MA.Mon3.spare0305 := FALSE;
   A_3125_MXZ02MA.Mon3.InReport := FALSE;
   A_3125_MXZ02MA.Mon3.OutTimeoutTime := FALSE;
   A_3125_MXZ02MA.Mon3.InHWStop := FALSE;
   A_3125_MXZ02MA.Mon3.InDPFault := FALSE;
   A_3125_MXZ02MA.Mon3.OutPreAlarmTrue := FALSE;
   A_3125_MXZ02MA.Mon3.OutPreAlarmFalse := FALSE;
   A_3125_MXZ02MA.Mon3.OutFlagPos := FALSE;
   A_3125_MXZ02MA.Mon3.OutFlagNeg := FALSE;
   A_3125_MXZ02MA.Mon3.OutpFaultReset := FALSE;
   A_3125_MXZ02MA.Mon3.OutTrue := FALSE;
   A_3125_MXZ02MA.Mon3.StFalse := FALSE;
   A_3125_MXZ02MA.Mon3.StCtoTrue := FALSE;
   A_3125_MXZ02MA.Mon3.StTrue := FALSE;
   A_3125_MXZ02MA.Mon3.StCtoFalse := FALSE;
   A_3125_MXZ02MA.Mon3.StFault := FALSE;
   A_3125_MXZ02MA.Mon3.OutAlarmNrLog := 0;
   A_3125_MXZ02MA.Mon3.Par.ParObjectNo := 0;
   A_3125_MXZ02MA.Mon3.Par.ParMsgType := 0;
   A_3125_MXZ02MA.Mon3.Par.ParHornCode := 0;
   A_3125_MXZ02MA.Mon3.Par.ParLogOff := FALSE;
   A_3125_MXZ02MA.Mon3.Par.spare0401 := FALSE;
   A_3125_MXZ02MA.Mon3.Par.Par2WorkingCond := FALSE;
   A_3125_MXZ02MA.Mon3.Par.ParFaultRetry := FALSE;
   A_3125_MXZ02MA.Mon3.Par.ParBinLevel := FALSE;
   A_3125_MXZ02MA.Mon3.Par.ParDelayChange := 0;
   A_3125_MXZ02MA.Mon3.Par.ParDelayTrue := 0;
   A_3125_MXZ02MA.Mon3.Par.ParDelayFalse := 0;
   A_3125_MXZ02MA.Mon3.Par.ParTimeoutTrue := 0;
   A_3125_MXZ02MA.Mon3.Par.ParTimeoutFalse := 0;
   A_3125_MXZ02MA.Mon3.Par.OutMonTime := 0;
   A_3125_MXZ02MA.Mon3.Par.OutTransitionTime := 0;
   A_3125_MXZ02MA.Mon3.Par.OutMonTrue := FALSE;
   A_3125_MXZ02MA.Mon3.Par.OutMonFalse := FALSE;
   A_3125_MXZ02MA.Mon3.Par.OutFlagFaultDev := FALSE;
   A_3125_MXZ02MA.Mon3.Par.OutDelayTime := 0;
   A_3125_MXZ02MA.Mon4.StCode := 0;
   A_3125_MXZ02MA.Mon4.InMonTrue := FALSE;
   A_3125_MXZ02MA.Mon4.InMonFalse := FALSE;
   A_3125_MXZ02MA.Mon4.InPreAlarmTrue := FALSE;
   A_3125_MXZ02MA.Mon4.InPreAlarmFalse := FALSE;
   A_3125_MXZ02MA.Mon4.InStopTrueTime := FALSE;
   A_3125_MXZ02MA.Mon4.InStopFalseTime := FALSE;
   A_3125_MXZ02MA.Mon4.InpTrue := FALSE;
   A_3125_MXZ02MA.Mon4.InpFaultDev := FALSE;
   A_3125_MXZ02MA.Mon4.CmdRstTrueTime := FALSE;
   A_3125_MXZ02MA.Mon4.CmdRstFalseTime := FALSE;
   A_3125_MXZ02MA.Mon4.CmdRunTimeoutTime := FALSE;
   A_3125_MXZ02MA.Mon4.CmdFaultReset := FALSE;
   A_3125_MXZ02MA.Mon4.InLocal := FALSE;
   A_3125_MXZ02MA.Mon4.spare0305 := FALSE;
   A_3125_MXZ02MA.Mon4.InReport := FALSE;
   A_3125_MXZ02MA.Mon4.OutTimeoutTime := FALSE;
   A_3125_MXZ02MA.Mon4.InHWStop := FALSE;
   A_3125_MXZ02MA.Mon4.InDPFault := FALSE;
   A_3125_MXZ02MA.Mon4.OutPreAlarmTrue := FALSE;
   A_3125_MXZ02MA.Mon4.OutPreAlarmFalse := FALSE;
   A_3125_MXZ02MA.Mon4.OutFlagPos := FALSE;
   A_3125_MXZ02MA.Mon4.OutFlagNeg := FALSE;
   A_3125_MXZ02MA.Mon4.OutpFaultReset := FALSE;
   A_3125_MXZ02MA.Mon4.OutTrue := FALSE;
   A_3125_MXZ02MA.Mon4.StFalse := FALSE;
   A_3125_MXZ02MA.Mon4.StCtoTrue := FALSE;
   A_3125_MXZ02MA.Mon4.StTrue := FALSE;
   A_3125_MXZ02MA.Mon4.StCtoFalse := FALSE;
   A_3125_MXZ02MA.Mon4.StFault := FALSE;
   A_3125_MXZ02MA.Mon4.OutAlarmNrLog := 0;
   A_3125_MXZ02MA.Mon4.Par.ParObjectNo := 0;
   A_3125_MXZ02MA.Mon4.Par.ParMsgType := 0;
   A_3125_MXZ02MA.Mon4.Par.ParHornCode := 0;
   A_3125_MXZ02MA.Mon4.Par.ParLogOff := FALSE;
   A_3125_MXZ02MA.Mon4.Par.spare0401 := FALSE;
   A_3125_MXZ02MA.Mon4.Par.Par2WorkingCond := FALSE;
   A_3125_MXZ02MA.Mon4.Par.ParFaultRetry := FALSE;
   A_3125_MXZ02MA.Mon4.Par.ParBinLevel := FALSE;
   A_3125_MXZ02MA.Mon4.Par.ParDelayChange := 0;
   A_3125_MXZ02MA.Mon4.Par.ParDelayTrue := 0;
   A_3125_MXZ02MA.Mon4.Par.ParDelayFalse := 0;
   A_3125_MXZ02MA.Mon4.Par.ParTimeoutTrue := 0;
   A_3125_MXZ02MA.Mon4.Par.ParTimeoutFalse := 0;
   A_3125_MXZ02MA.Mon4.Par.OutMonTime := 0;
   A_3125_MXZ02MA.Mon4.Par.OutTransitionTime := 0;
   A_3125_MXZ02MA.Mon4.Par.OutMonTrue := FALSE;
   A_3125_MXZ02MA.Mon4.Par.OutMonFalse := FALSE;
   A_3125_MXZ02MA.Mon4.Par.OutFlagFaultDev := FALSE;
   A_3125_MXZ02MA.Mon4.Par.OutDelayTime := 0;
   A_3125_MXZ02MA.Mon5.StCode := 0;
   A_3125_MXZ02MA.Mon5.InMonTrue := FALSE;
   A_3125_MXZ02MA.Mon5.InMonFalse := FALSE;
   A_3125_MXZ02MA.Mon5.InPreAlarmTrue := FALSE;
   A_3125_MXZ02MA.Mon5.InPreAlarmFalse := FALSE;
   A_3125_MXZ02MA.Mon5.InStopTrueTime := FALSE;
   A_3125_MXZ02MA.Mon5.InStopFalseTime := FALSE;
   A_3125_MXZ02MA.Mon5.InpTrue := FALSE;
   A_3125_MXZ02MA.Mon5.InpFaultDev := FALSE;
   A_3125_MXZ02MA.Mon5.CmdRstTrueTime := FALSE;
   A_3125_MXZ02MA.Mon5.CmdRstFalseTime := FALSE;
   A_3125_MXZ02MA.Mon5.CmdRunTimeoutTime := FALSE;
   A_3125_MXZ02MA.Mon5.CmdFaultReset := FALSE;
   A_3125_MXZ02MA.Mon5.InLocal := FALSE;
   A_3125_MXZ02MA.Mon5.spare0305 := FALSE;
   A_3125_MXZ02MA.Mon5.InReport := FALSE;
   A_3125_MXZ02MA.Mon5.OutTimeoutTime := FALSE;
   A_3125_MXZ02MA.Mon5.InHWStop := FALSE;
   A_3125_MXZ02MA.Mon5.InDPFault := FALSE;
   A_3125_MXZ02MA.Mon5.OutPreAlarmTrue := FALSE;
   A_3125_MXZ02MA.Mon5.OutPreAlarmFalse := FALSE;
   A_3125_MXZ02MA.Mon5.OutFlagPos := FALSE;
   A_3125_MXZ02MA.Mon5.OutFlagNeg := FALSE;
   A_3125_MXZ02MA.Mon5.OutpFaultReset := FALSE;
   A_3125_MXZ02MA.Mon5.OutTrue := FALSE;
   A_3125_MXZ02MA.Mon5.StFalse := FALSE;
   A_3125_MXZ02MA.Mon5.StCtoTrue := FALSE;
   A_3125_MXZ02MA.Mon5.StTrue := FALSE;
   A_3125_MXZ02MA.Mon5.StCtoFalse := FALSE;
   A_3125_MXZ02MA.Mon5.StFault := FALSE;
   A_3125_MXZ02MA.Mon5.OutAlarmNrLog := 0;
   A_3125_MXZ02MA.Mon5.Par.ParObjectNo := 0;
   A_3125_MXZ02MA.Mon5.Par.ParMsgType := 0;
   A_3125_MXZ02MA.Mon5.Par.ParHornCode := 0;
   A_3125_MXZ02MA.Mon5.Par.ParLogOff := FALSE;
   A_3125_MXZ02MA.Mon5.Par.spare0401 := FALSE;
   A_3125_MXZ02MA.Mon5.Par.Par2WorkingCond := FALSE;
   A_3125_MXZ02MA.Mon5.Par.ParFaultRetry := FALSE;
   A_3125_MXZ02MA.Mon5.Par.ParBinLevel := FALSE;
   A_3125_MXZ02MA.Mon5.Par.ParDelayChange := 0;
   A_3125_MXZ02MA.Mon5.Par.ParDelayTrue := 0;
   A_3125_MXZ02MA.Mon5.Par.ParDelayFalse := 0;
   A_3125_MXZ02MA.Mon5.Par.ParTimeoutTrue := 0;
   A_3125_MXZ02MA.Mon5.Par.ParTimeoutFalse := 0;
   A_3125_MXZ02MA.Mon5.Par.OutMonTime := 0;
   A_3125_MXZ02MA.Mon5.Par.OutTransitionTime := 0;
   A_3125_MXZ02MA.Mon5.Par.OutMonTrue := FALSE;
   A_3125_MXZ02MA.Mon5.Par.OutMonFalse := FALSE;
   A_3125_MXZ02MA.Mon5.Par.OutFlagFaultDev := FALSE;
   A_3125_MXZ02MA.Mon5.Par.OutDelayTime := 0;
   A_3125_MXZ02MA.Mon6.StCode := 0;
   A_3125_MXZ02MA.Mon6.InMonTrue := FALSE;
   A_3125_MXZ02MA.Mon6.InMonFalse := FALSE;
   A_3125_MXZ02MA.Mon6.InPreAlarmTrue := FALSE;
   A_3125_MXZ02MA.Mon6.InPreAlarmFalse := FALSE;
   A_3125_MXZ02MA.Mon6.InStopTrueTime := FALSE;
   A_3125_MXZ02MA.Mon6.InStopFalseTime := FALSE;
   A_3125_MXZ02MA.Mon6.InpTrue := FALSE;
   A_3125_MXZ02MA.Mon6.InpFaultDev := FALSE;
   A_3125_MXZ02MA.Mon6.CmdRstTrueTime := FALSE;
   A_3125_MXZ02MA.Mon6.CmdRstFalseTime := FALSE;
   A_3125_MXZ02MA.Mon6.CmdRunTimeoutTime := FALSE;
   A_3125_MXZ02MA.Mon6.CmdFaultReset := FALSE;
   A_3125_MXZ02MA.Mon6.InLocal := FALSE;
   A_3125_MXZ02MA.Mon6.spare0305 := FALSE;
   A_3125_MXZ02MA.Mon6.InReport := FALSE;
   A_3125_MXZ02MA.Mon6.OutTimeoutTime := FALSE;
   A_3125_MXZ02MA.Mon6.InHWStop := FALSE;
   A_3125_MXZ02MA.Mon6.InDPFault := FALSE;
   A_3125_MXZ02MA.Mon6.OutPreAlarmTrue := FALSE;
   A_3125_MXZ02MA.Mon6.OutPreAlarmFalse := FALSE;
   A_3125_MXZ02MA.Mon6.OutFlagPos := FALSE;
   A_3125_MXZ02MA.Mon6.OutFlagNeg := FALSE;
   A_3125_MXZ02MA.Mon6.OutpFaultReset := FALSE;
   A_3125_MXZ02MA.Mon6.OutTrue := FALSE;
   A_3125_MXZ02MA.Mon6.StFalse := FALSE;
   A_3125_MXZ02MA.Mon6.StCtoTrue := FALSE;
   A_3125_MXZ02MA.Mon6.StTrue := FALSE;
   A_3125_MXZ02MA.Mon6.StCtoFalse := FALSE;
   A_3125_MXZ02MA.Mon6.StFault := FALSE;
   A_3125_MXZ02MA.Mon6.OutAlarmNrLog := 0;
   A_3125_MXZ02MA.Mon6.Par.ParObjectNo := 0;
   A_3125_MXZ02MA.Mon6.Par.ParMsgType := 0;
   A_3125_MXZ02MA.Mon6.Par.ParHornCode := 0;
   A_3125_MXZ02MA.Mon6.Par.ParLogOff := FALSE;
   A_3125_MXZ02MA.Mon6.Par.spare0401 := FALSE;
   A_3125_MXZ02MA.Mon6.Par.Par2WorkingCond := FALSE;
   A_3125_MXZ02MA.Mon6.Par.ParFaultRetry := FALSE;
   A_3125_MXZ02MA.Mon6.Par.ParBinLevel := FALSE;
   A_3125_MXZ02MA.Mon6.Par.ParDelayChange := 0;
   A_3125_MXZ02MA.Mon6.Par.ParDelayTrue := 0;
   A_3125_MXZ02MA.Mon6.Par.ParDelayFalse := 0;
   A_3125_MXZ02MA.Mon6.Par.ParTimeoutTrue := 0;
   A_3125_MXZ02MA.Mon6.Par.ParTimeoutFalse := 0;
   A_3125_MXZ02MA.Mon6.Par.OutMonTime := 0;
   A_3125_MXZ02MA.Mon6.Par.OutTransitionTime := 0;
   A_3125_MXZ02MA.Mon6.Par.OutMonTrue := FALSE;
   A_3125_MXZ02MA.Mon6.Par.OutMonFalse := FALSE;
   A_3125_MXZ02MA.Mon6.Par.OutFlagFaultDev := FALSE;
   A_3125_MXZ02MA.Mon6.Par.OutDelayTime := 0;
   A_3125_MXZ02MA.A_3125_MXZ02.StCode := 0;
   A_3125_MXZ02MA.A_3125_MXZ02.InEnableRev := FALSE;
   A_3125_MXZ02MA.A_3125_MXZ02.InEnableFwd := FALSE;
   A_3125_MXZ02MA.A_3125_MXZ02.InSlow := FALSE;
   A_3125_MXZ02MA.A_3125_MXZ02.InpRunSlow := FALSE;
   A_3125_MXZ02MA.A_3125_MXZ02.InpRunFast := FALSE;
   A_3125_MXZ02MA.A_3125_MXZ02.InpRunRev := FALSE;
   A_3125_MXZ02MA.A_3125_MXZ02.InpRunFwd := FALSE;
   A_3125_MXZ02MA.A_3125_MXZ02.InpFaultDev := FALSE;
   A_3125_MXZ02MA.A_3125_MXZ02.CmdOff := FALSE;
   A_3125_MXZ02MA.A_3125_MXZ02.CmdOn := FALSE;
   A_3125_MXZ02MA.A_3125_MXZ02.CmdNext := FALSE;
   A_3125_MXZ02MA.A_3125_MXZ02.CmdFaultReset := FALSE;
   A_3125_MXZ02MA.A_3125_MXZ02.InLocal := FALSE;
   A_3125_MXZ02MA.A_3125_MXZ02.InManual := FALSE;
   A_3125_MXZ02MA.A_3125_MXZ02.InReport := FALSE;
   A_3125_MXZ02MA.A_3125_MXZ02.InSeqStop := FALSE;
   A_3125_MXZ02MA.A_3125_MXZ02.InHWStop := FALSE;
   A_3125_MXZ02MA.A_3125_MXZ02.InDPFault := FALSE;
   A_3125_MXZ02MA.A_3125_MXZ02.OutIdling := FALSE;
   A_3125_MXZ02MA.A_3125_MXZ02.OutpRunSlow := FALSE;
   A_3125_MXZ02MA.A_3125_MXZ02.OutpRunFast := FALSE;
   A_3125_MXZ02MA.A_3125_MXZ02.OutpRunRev := FALSE;
   A_3125_MXZ02MA.A_3125_MXZ02.OutpRunFwd := FALSE;
   A_3125_MXZ02MA.A_3125_MXZ02.OutpFaultReset := FALSE;
   A_3125_MXZ02MA.A_3125_MXZ02.StStopped := FALSE;
   A_3125_MXZ02MA.A_3125_MXZ02.StStarting := FALSE;
   A_3125_MXZ02MA.A_3125_MXZ02.StStartedFwd := FALSE;
   A_3125_MXZ02MA.A_3125_MXZ02.StStopping := FALSE;
   A_3125_MXZ02MA.A_3125_MXZ02.StFault := FALSE;
   A_3125_MXZ02MA.A_3125_MXZ02.StStartedRev := FALSE;
   A_3125_MXZ02MA.A_3125_MXZ02.InOutManSlow := FALSE;
   A_3125_MXZ02MA.A_3125_MXZ02.InOutManRev := FALSE;
   A_3125_MXZ02MA.A_3125_MXZ02.OutAlarmNrLog := 0;
   A_3125_MXZ02MA.A_3125_MXZ02.Par.ParObjectNo := 27129;
   A_3125_MXZ02MA.A_3125_MXZ02.Par.ParMsgType := 7053;
   A_3125_MXZ02MA.A_3125_MXZ02.Par.ParHornCode := 1;
   A_3125_MXZ02MA.A_3125_MXZ02.Par.ParLogOff := FALSE;
   A_3125_MXZ02MA.A_3125_MXZ02.Par.ParManual := TRUE;
   A_3125_MXZ02MA.A_3125_MXZ02.Par.ParRestartDelay := FALSE;
   A_3125_MXZ02MA.A_3125_MXZ02.Par.Par2Speed := FALSE;
   A_3125_MXZ02MA.A_3125_MXZ02.Par.ParHeavyStartup := FALSE;
   A_3125_MXZ02MA.A_3125_MXZ02.Par.spare45 := FALSE;
   A_3125_MXZ02MA.A_3125_MXZ02.Par.spare46 := FALSE;
   A_3125_MXZ02MA.A_3125_MXZ02.Par.OutEdgeFaultReset := FALSE;
   A_3125_MXZ02MA.A_3125_MXZ02.Par.OutDelayFault := FALSE;
   A_3125_MXZ02MA.A_3125_MXZ02.Par.OutFlagFaultDev := FALSE;
   A_3125_MXZ02MA.A_3125_MXZ02.Par.ParMonTime := 20;
   A_3125_MXZ02MA.A_3125_MXZ02.Par.ParStartingTime := 20;
   A_3125_MXZ02MA.A_3125_MXZ02.Par.ParStoppingTime := 0;
   A_3125_MXZ02MA.A_3125_MXZ02.Par.ParIdlingTime := 0;
   A_3125_MXZ02MA.A_3125_MXZ02.Par.ParDelayTime := 10;
   A_3125_MXZ02MA.A_3125_MXZ02.Par.OutMonTime := 0;
   A_3125_MXZ02MA.A_3125_MXZ02.Par.OutTransitionTime := 0;
   A_3125_MXZ02MA.A_3125_MXZ02.Par.OutDelayTime := 0;
   A_3125_MXZ02MA.A_3125_MXZ02.Par.InOutManPulseLen := 0;
   A_3126_MXZ02MA.Ma.StCode := 0;
   A_3126_MXZ02MA.Ma.InEnableRev := FALSE;
   A_3126_MXZ02MA.Ma.InEnableFwd := FALSE;
   A_3126_MXZ02MA.Ma.InOverrideHLOutlet := FALSE;
   A_3126_MXZ02MA.Ma.spare0203 := FALSE;
   A_3126_MXZ02MA.Ma.OutEdgeFaultReset := FALSE;
   A_3126_MXZ02MA.Ma.OutFaultResetFcttst := FALSE;
   A_3126_MXZ02MA.Ma.InpControlEBM := FALSE;
   A_3126_MXZ02MA.Ma.InpLocked := FALSE;
   A_3126_MXZ02MA.Ma.CmdOff := FALSE;
   A_3126_MXZ02MA.Ma.CmdOn := FALSE;
   A_3126_MXZ02MA.Ma.CmdNext := FALSE;
   A_3126_MXZ02MA.Ma.CmdFaultReset := FALSE;
   A_3126_MXZ02MA.Ma.InLocal := FALSE;
   A_3126_MXZ02MA.Ma.InManual := FALSE;
   A_3126_MXZ02MA.Ma.CmdTestEBM := FALSE;
   A_3126_MXZ02MA.Ma.InSeqStop := FALSE;
   A_3126_MXZ02MA.Ma.OutWarning := FALSE;
   A_3126_MXZ02MA.Ma.InfBMTopOk := FALSE;
   A_3126_MXZ02MA.Ma.InfBMBottomOk := FALSE;
   A_3126_MXZ02MA.Ma.InfSMOk := FALSE;
   A_3126_MXZ02MA.Ma.OutpFcttst_BM_Top := FALSE;
   A_3126_MXZ02MA.Ma.OutpFcttst_BM_Bottom := FALSE;
   A_3126_MXZ02MA.Ma.OutpFcttst_SM := FALSE;
   A_3126_MXZ02MA.Ma.OutpFaultReset := FALSE;
   A_3126_MXZ02MA.Ma.StStopped := FALSE;
   A_3126_MXZ02MA.Ma.StStarting := FALSE;
   A_3126_MXZ02MA.Ma.StStartedFwd := FALSE;
   A_3126_MXZ02MA.Ma.StStopping := FALSE;
   A_3126_MXZ02MA.Ma.StFault := FALSE;
   A_3126_MXZ02MA.Ma.StStartedRev := FALSE;
   A_3126_MXZ02MA.Ma.StLocked := FALSE;
   A_3126_MXZ02MA.Ma.OutTestTime := 0;
   A_3126_MXZ02MA.Ma.Par.ParObjectNo := 27131;
   A_3126_MXZ02MA.Ma.Par.ParWithMon1 := TRUE;
   A_3126_MXZ02MA.Ma.Par.ParWithMon3 := FALSE;
   A_3126_MXZ02MA.Ma.Par.ParWithMon4 := FALSE;
   A_3126_MXZ02MA.Ma.Par.ParWithMon5 := FALSE;
   A_3126_MXZ02MA.Ma.Par.ParWithMon6 := FALSE;
   A_3126_MXZ02MA.Ma.Par.ParMon1IsHL := FALSE;
   A_3126_MXZ02MA.Ma.Par.ParMon1IsLS := TRUE;
   A_3126_MXZ02MA.Ma.Par.ParMon1StopByFault := TRUE;
   A_3126_MXZ02MA.Ma.Par.ParMon2IsLS := FALSE;
   A_3126_MXZ02MA.Ma.Par.ParMon3IsLS := FALSE;
   A_3126_MXZ02MA.Ma.Par.ParMon4AsWarning := FALSE;
   A_3126_MXZ02MA.Ma.Par.ParMon4StopByFault := FALSE;
   A_3126_MXZ02MA.Ma.Par.ParMon4IsLS := FALSE;
   A_3126_MXZ02MA.Ma.Par.ParEBM := FALSE;
   A_3126_MXZ02MA.Ma.Par.ParMon4IsSM := FALSE;
   A_3126_MXZ02MA.A_3225_BFT09.StCode := 0;
   A_3126_MXZ02MA.A_3225_BFT09.InMonTrue := FALSE;
   A_3126_MXZ02MA.A_3225_BFT09.InMonFalse := FALSE;
   A_3126_MXZ02MA.A_3225_BFT09.InPreAlarmTrue := FALSE;
   A_3126_MXZ02MA.A_3225_BFT09.InPreAlarmFalse := FALSE;
   A_3126_MXZ02MA.A_3225_BFT09.InStopTrueTime := FALSE;
   A_3126_MXZ02MA.A_3225_BFT09.InStopFalseTime := FALSE;
   A_3126_MXZ02MA.A_3225_BFT09.InpTrue := FALSE;
   A_3126_MXZ02MA.A_3225_BFT09.InpFaultDev := FALSE;
   A_3126_MXZ02MA.A_3225_BFT09.CmdRstTrueTime := FALSE;
   A_3126_MXZ02MA.A_3225_BFT09.CmdRstFalseTime := FALSE;
   A_3126_MXZ02MA.A_3225_BFT09.CmdRunTimeoutTime := FALSE;
   A_3126_MXZ02MA.A_3225_BFT09.CmdFaultReset := FALSE;
   A_3126_MXZ02MA.A_3225_BFT09.InLocal := FALSE;
   A_3126_MXZ02MA.A_3225_BFT09.spare0305 := FALSE;
   A_3126_MXZ02MA.A_3225_BFT09.InReport := FALSE;
   A_3126_MXZ02MA.A_3225_BFT09.OutTimeoutTime := FALSE;
   A_3126_MXZ02MA.A_3225_BFT09.InHWStop := FALSE;
   A_3126_MXZ02MA.A_3225_BFT09.InDPFault := FALSE;
   A_3126_MXZ02MA.A_3225_BFT09.OutPreAlarmTrue := FALSE;
   A_3126_MXZ02MA.A_3225_BFT09.OutPreAlarmFalse := FALSE;
   A_3126_MXZ02MA.A_3225_BFT09.OutFlagPos := FALSE;
   A_3126_MXZ02MA.A_3225_BFT09.OutFlagNeg := FALSE;
   A_3126_MXZ02MA.A_3225_BFT09.OutpFaultReset := FALSE;
   A_3126_MXZ02MA.A_3225_BFT09.OutTrue := FALSE;
   A_3126_MXZ02MA.A_3225_BFT09.StFalse := FALSE;
   A_3126_MXZ02MA.A_3225_BFT09.StCtoTrue := FALSE;
   A_3126_MXZ02MA.A_3225_BFT09.StTrue := FALSE;
   A_3126_MXZ02MA.A_3225_BFT09.StCtoFalse := FALSE;
   A_3126_MXZ02MA.A_3225_BFT09.StFault := FALSE;
   A_3126_MXZ02MA.A_3225_BFT09.OutAlarmNrLog := 0;
   A_3126_MXZ02MA.A_3225_BFT09.Par.ParObjectNo := 27132;
   A_3126_MXZ02MA.A_3225_BFT09.Par.ParMsgType := 7135;
   A_3126_MXZ02MA.A_3225_BFT09.Par.ParHornCode := 0;
   A_3126_MXZ02MA.A_3225_BFT09.Par.ParLogOff := FALSE;
   A_3126_MXZ02MA.A_3225_BFT09.Par.spare0401 := FALSE;
   A_3126_MXZ02MA.A_3225_BFT09.Par.Par2WorkingCond := FALSE;
   A_3126_MXZ02MA.A_3225_BFT09.Par.ParFaultRetry := FALSE;
   A_3126_MXZ02MA.A_3225_BFT09.Par.ParBinLevel := FALSE;
   A_3126_MXZ02MA.A_3225_BFT09.Par.ParDelayChange := 0;
   A_3126_MXZ02MA.A_3225_BFT09.Par.ParDelayTrue := 10;
   A_3126_MXZ02MA.A_3225_BFT09.Par.ParDelayFalse := 0;
   A_3126_MXZ02MA.A_3225_BFT09.Par.ParTimeoutTrue := 0;
   A_3126_MXZ02MA.A_3225_BFT09.Par.ParTimeoutFalse := 0;
   A_3126_MXZ02MA.A_3225_BFT09.Par.OutMonTime := 0;
   A_3126_MXZ02MA.A_3225_BFT09.Par.OutTransitionTime := 0;
   A_3126_MXZ02MA.A_3225_BFT09.Par.OutMonTrue := FALSE;
   A_3126_MXZ02MA.A_3225_BFT09.Par.OutMonFalse := FALSE;
   A_3126_MXZ02MA.A_3225_BFT09.Par.OutFlagFaultDev := FALSE;
   A_3126_MXZ02MA.A_3225_BFT09.Par.OutDelayTime := 0;
   A_3126_MXZ02MA.Mon2.StCode := 0;
   A_3126_MXZ02MA.Mon2.InMonTrue := FALSE;
   A_3126_MXZ02MA.Mon2.InMonFalse := FALSE;
   A_3126_MXZ02MA.Mon2.InPreAlarmTrue := FALSE;
   A_3126_MXZ02MA.Mon2.InPreAlarmFalse := FALSE;
   A_3126_MXZ02MA.Mon2.InStopTrueTime := FALSE;
   A_3126_MXZ02MA.Mon2.InStopFalseTime := FALSE;
   A_3126_MXZ02MA.Mon2.InpTrue := FALSE;
   A_3126_MXZ02MA.Mon2.InpFaultDev := FALSE;
   A_3126_MXZ02MA.Mon2.CmdRstTrueTime := FALSE;
   A_3126_MXZ02MA.Mon2.CmdRstFalseTime := FALSE;
   A_3126_MXZ02MA.Mon2.CmdRunTimeoutTime := FALSE;
   A_3126_MXZ02MA.Mon2.CmdFaultReset := FALSE;
   A_3126_MXZ02MA.Mon2.InLocal := FALSE;
   A_3126_MXZ02MA.Mon2.spare0305 := FALSE;
   A_3126_MXZ02MA.Mon2.InReport := FALSE;
   A_3126_MXZ02MA.Mon2.OutTimeoutTime := FALSE;
   A_3126_MXZ02MA.Mon2.InHWStop := FALSE;
   A_3126_MXZ02MA.Mon2.InDPFault := FALSE;
   A_3126_MXZ02MA.Mon2.OutPreAlarmTrue := FALSE;
   A_3126_MXZ02MA.Mon2.OutPreAlarmFalse := FALSE;
   A_3126_MXZ02MA.Mon2.OutFlagPos := FALSE;
   A_3126_MXZ02MA.Mon2.OutFlagNeg := FALSE;
   A_3126_MXZ02MA.Mon2.OutpFaultReset := FALSE;
   A_3126_MXZ02MA.Mon2.OutTrue := FALSE;
   A_3126_MXZ02MA.Mon2.StFalse := FALSE;
   A_3126_MXZ02MA.Mon2.StCtoTrue := FALSE;
   A_3126_MXZ02MA.Mon2.StTrue := FALSE;
   A_3126_MXZ02MA.Mon2.StCtoFalse := FALSE;
   A_3126_MXZ02MA.Mon2.StFault := FALSE;
   A_3126_MXZ02MA.Mon2.OutAlarmNrLog := 0;
   A_3126_MXZ02MA.Mon2.Par.ParObjectNo := 0;
   A_3126_MXZ02MA.Mon2.Par.ParMsgType := 0;
   A_3126_MXZ02MA.Mon2.Par.ParHornCode := 0;
   A_3126_MXZ02MA.Mon2.Par.ParLogOff := FALSE;
   A_3126_MXZ02MA.Mon2.Par.spare0401 := FALSE;
   A_3126_MXZ02MA.Mon2.Par.Par2WorkingCond := FALSE;
   A_3126_MXZ02MA.Mon2.Par.ParFaultRetry := FALSE;
   A_3126_MXZ02MA.Mon2.Par.ParBinLevel := FALSE;
   A_3126_MXZ02MA.Mon2.Par.ParDelayChange := 0;
   A_3126_MXZ02MA.Mon2.Par.ParDelayTrue := 0;
   A_3126_MXZ02MA.Mon2.Par.ParDelayFalse := 0;
   A_3126_MXZ02MA.Mon2.Par.ParTimeoutTrue := 0;
   A_3126_MXZ02MA.Mon2.Par.ParTimeoutFalse := 0;
   A_3126_MXZ02MA.Mon2.Par.OutMonTime := 0;
   A_3126_MXZ02MA.Mon2.Par.OutTransitionTime := 0;
   A_3126_MXZ02MA.Mon2.Par.OutMonTrue := FALSE;
   A_3126_MXZ02MA.Mon2.Par.OutMonFalse := FALSE;
   A_3126_MXZ02MA.Mon2.Par.OutFlagFaultDev := FALSE;
   A_3126_MXZ02MA.Mon2.Par.OutDelayTime := 0;
   A_3126_MXZ02MA.Mon3.StCode := 0;
   A_3126_MXZ02MA.Mon3.InMonTrue := FALSE;
   A_3126_MXZ02MA.Mon3.InMonFalse := FALSE;
   A_3126_MXZ02MA.Mon3.InPreAlarmTrue := FALSE;
   A_3126_MXZ02MA.Mon3.InPreAlarmFalse := FALSE;
   A_3126_MXZ02MA.Mon3.InStopTrueTime := FALSE;
   A_3126_MXZ02MA.Mon3.InStopFalseTime := FALSE;
   A_3126_MXZ02MA.Mon3.InpTrue := FALSE;
   A_3126_MXZ02MA.Mon3.InpFaultDev := FALSE;
   A_3126_MXZ02MA.Mon3.CmdRstTrueTime := FALSE;
   A_3126_MXZ02MA.Mon3.CmdRstFalseTime := FALSE;
   A_3126_MXZ02MA.Mon3.CmdRunTimeoutTime := FALSE;
   A_3126_MXZ02MA.Mon3.CmdFaultReset := FALSE;
   A_3126_MXZ02MA.Mon3.InLocal := FALSE;
   A_3126_MXZ02MA.Mon3.spare0305 := FALSE;
   A_3126_MXZ02MA.Mon3.InReport := FALSE;
   A_3126_MXZ02MA.Mon3.OutTimeoutTime := FALSE;
   A_3126_MXZ02MA.Mon3.InHWStop := FALSE;
   A_3126_MXZ02MA.Mon3.InDPFault := FALSE;
   A_3126_MXZ02MA.Mon3.OutPreAlarmTrue := FALSE;
   A_3126_MXZ02MA.Mon3.OutPreAlarmFalse := FALSE;
   A_3126_MXZ02MA.Mon3.OutFlagPos := FALSE;
   A_3126_MXZ02MA.Mon3.OutFlagNeg := FALSE;
   A_3126_MXZ02MA.Mon3.OutpFaultReset := FALSE;
   A_3126_MXZ02MA.Mon3.OutTrue := FALSE;
   A_3126_MXZ02MA.Mon3.StFalse := FALSE;
   A_3126_MXZ02MA.Mon3.StCtoTrue := FALSE;
   A_3126_MXZ02MA.Mon3.StTrue := FALSE;
   A_3126_MXZ02MA.Mon3.StCtoFalse := FALSE;
   A_3126_MXZ02MA.Mon3.StFault := FALSE;
   A_3126_MXZ02MA.Mon3.OutAlarmNrLog := 0;
   A_3126_MXZ02MA.Mon3.Par.ParObjectNo := 0;
   A_3126_MXZ02MA.Mon3.Par.ParMsgType := 0;
   A_3126_MXZ02MA.Mon3.Par.ParHornCode := 0;
   A_3126_MXZ02MA.Mon3.Par.ParLogOff := FALSE;
   A_3126_MXZ02MA.Mon3.Par.spare0401 := FALSE;
   A_3126_MXZ02MA.Mon3.Par.Par2WorkingCond := FALSE;
   A_3126_MXZ02MA.Mon3.Par.ParFaultRetry := FALSE;
   A_3126_MXZ02MA.Mon3.Par.ParBinLevel := FALSE;
   A_3126_MXZ02MA.Mon3.Par.ParDelayChange := 0;
   A_3126_MXZ02MA.Mon3.Par.ParDelayTrue := 0;
   A_3126_MXZ02MA.Mon3.Par.ParDelayFalse := 0;
   A_3126_MXZ02MA.Mon3.Par.ParTimeoutTrue := 0;
   A_3126_MXZ02MA.Mon3.Par.ParTimeoutFalse := 0;
   A_3126_MXZ02MA.Mon3.Par.OutMonTime := 0;
   A_3126_MXZ02MA.Mon3.Par.OutTransitionTime := 0;
   A_3126_MXZ02MA.Mon3.Par.OutMonTrue := FALSE;
   A_3126_MXZ02MA.Mon3.Par.OutMonFalse := FALSE;
   A_3126_MXZ02MA.Mon3.Par.OutFlagFaultDev := FALSE;
   A_3126_MXZ02MA.Mon3.Par.OutDelayTime := 0;
   A_3126_MXZ02MA.Mon4.StCode := 0;
   A_3126_MXZ02MA.Mon4.InMonTrue := FALSE;
   A_3126_MXZ02MA.Mon4.InMonFalse := FALSE;
   A_3126_MXZ02MA.Mon4.InPreAlarmTrue := FALSE;
   A_3126_MXZ02MA.Mon4.InPreAlarmFalse := FALSE;
   A_3126_MXZ02MA.Mon4.InStopTrueTime := FALSE;
   A_3126_MXZ02MA.Mon4.InStopFalseTime := FALSE;
   A_3126_MXZ02MA.Mon4.InpTrue := FALSE;
   A_3126_MXZ02MA.Mon4.InpFaultDev := FALSE;
   A_3126_MXZ02MA.Mon4.CmdRstTrueTime := FALSE;
   A_3126_MXZ02MA.Mon4.CmdRstFalseTime := FALSE;
   A_3126_MXZ02MA.Mon4.CmdRunTimeoutTime := FALSE;
   A_3126_MXZ02MA.Mon4.CmdFaultReset := FALSE;
   A_3126_MXZ02MA.Mon4.InLocal := FALSE;
   A_3126_MXZ02MA.Mon4.spare0305 := FALSE;
   A_3126_MXZ02MA.Mon4.InReport := FALSE;
   A_3126_MXZ02MA.Mon4.OutTimeoutTime := FALSE;
   A_3126_MXZ02MA.Mon4.InHWStop := FALSE;
   A_3126_MXZ02MA.Mon4.InDPFault := FALSE;
   A_3126_MXZ02MA.Mon4.OutPreAlarmTrue := FALSE;
   A_3126_MXZ02MA.Mon4.OutPreAlarmFalse := FALSE;
   A_3126_MXZ02MA.Mon4.OutFlagPos := FALSE;
   A_3126_MXZ02MA.Mon4.OutFlagNeg := FALSE;
   A_3126_MXZ02MA.Mon4.OutpFaultReset := FALSE;
   A_3126_MXZ02MA.Mon4.OutTrue := FALSE;
   A_3126_MXZ02MA.Mon4.StFalse := FALSE;
   A_3126_MXZ02MA.Mon4.StCtoTrue := FALSE;
   A_3126_MXZ02MA.Mon4.StTrue := FALSE;
   A_3126_MXZ02MA.Mon4.StCtoFalse := FALSE;
   A_3126_MXZ02MA.Mon4.StFault := FALSE;
   A_3126_MXZ02MA.Mon4.OutAlarmNrLog := 0;
   A_3126_MXZ02MA.Mon4.Par.ParObjectNo := 0;
   A_3126_MXZ02MA.Mon4.Par.ParMsgType := 0;
   A_3126_MXZ02MA.Mon4.Par.ParHornCode := 0;
   A_3126_MXZ02MA.Mon4.Par.ParLogOff := FALSE;
   A_3126_MXZ02MA.Mon4.Par.spare0401 := FALSE;
   A_3126_MXZ02MA.Mon4.Par.Par2WorkingCond := FALSE;
   A_3126_MXZ02MA.Mon4.Par.ParFaultRetry := FALSE;
   A_3126_MXZ02MA.Mon4.Par.ParBinLevel := FALSE;
   A_3126_MXZ02MA.Mon4.Par.ParDelayChange := 0;
   A_3126_MXZ02MA.Mon4.Par.ParDelayTrue := 0;
   A_3126_MXZ02MA.Mon4.Par.ParDelayFalse := 0;
   A_3126_MXZ02MA.Mon4.Par.ParTimeoutTrue := 0;
   A_3126_MXZ02MA.Mon4.Par.ParTimeoutFalse := 0;
   A_3126_MXZ02MA.Mon4.Par.OutMonTime := 0;
   A_3126_MXZ02MA.Mon4.Par.OutTransitionTime := 0;
   A_3126_MXZ02MA.Mon4.Par.OutMonTrue := FALSE;
   A_3126_MXZ02MA.Mon4.Par.OutMonFalse := FALSE;
   A_3126_MXZ02MA.Mon4.Par.OutFlagFaultDev := FALSE;
   A_3126_MXZ02MA.Mon4.Par.OutDelayTime := 0;
   A_3126_MXZ02MA.Mon5.StCode := 0;
   A_3126_MXZ02MA.Mon5.InMonTrue := FALSE;
   A_3126_MXZ02MA.Mon5.InMonFalse := FALSE;
   A_3126_MXZ02MA.Mon5.InPreAlarmTrue := FALSE;
   A_3126_MXZ02MA.Mon5.InPreAlarmFalse := FALSE;
   A_3126_MXZ02MA.Mon5.InStopTrueTime := FALSE;
   A_3126_MXZ02MA.Mon5.InStopFalseTime := FALSE;
   A_3126_MXZ02MA.Mon5.InpTrue := FALSE;
   A_3126_MXZ02MA.Mon5.InpFaultDev := FALSE;
   A_3126_MXZ02MA.Mon5.CmdRstTrueTime := FALSE;
   A_3126_MXZ02MA.Mon5.CmdRstFalseTime := FALSE;
   A_3126_MXZ02MA.Mon5.CmdRunTimeoutTime := FALSE;
   A_3126_MXZ02MA.Mon5.CmdFaultReset := FALSE;
   A_3126_MXZ02MA.Mon5.InLocal := FALSE;
   A_3126_MXZ02MA.Mon5.spare0305 := FALSE;
   A_3126_MXZ02MA.Mon5.InReport := FALSE;
   A_3126_MXZ02MA.Mon5.OutTimeoutTime := FALSE;
   A_3126_MXZ02MA.Mon5.InHWStop := FALSE;
   A_3126_MXZ02MA.Mon5.InDPFault := FALSE;
   A_3126_MXZ02MA.Mon5.OutPreAlarmTrue := FALSE;
   A_3126_MXZ02MA.Mon5.OutPreAlarmFalse := FALSE;
   A_3126_MXZ02MA.Mon5.OutFlagPos := FALSE;
   A_3126_MXZ02MA.Mon5.OutFlagNeg := FALSE;
   A_3126_MXZ02MA.Mon5.OutpFaultReset := FALSE;
   A_3126_MXZ02MA.Mon5.OutTrue := FALSE;
   A_3126_MXZ02MA.Mon5.StFalse := FALSE;
   A_3126_MXZ02MA.Mon5.StCtoTrue := FALSE;
   A_3126_MXZ02MA.Mon5.StTrue := FALSE;
   A_3126_MXZ02MA.Mon5.StCtoFalse := FALSE;
   A_3126_MXZ02MA.Mon5.StFault := FALSE;
   A_3126_MXZ02MA.Mon5.OutAlarmNrLog := 0;
   A_3126_MXZ02MA.Mon5.Par.ParObjectNo := 0;
   A_3126_MXZ02MA.Mon5.Par.ParMsgType := 0;
   A_3126_MXZ02MA.Mon5.Par.ParHornCode := 0;
   A_3126_MXZ02MA.Mon5.Par.ParLogOff := FALSE;
   A_3126_MXZ02MA.Mon5.Par.spare0401 := FALSE;
   A_3126_MXZ02MA.Mon5.Par.Par2WorkingCond := FALSE;
   A_3126_MXZ02MA.Mon5.Par.ParFaultRetry := FALSE;
   A_3126_MXZ02MA.Mon5.Par.ParBinLevel := FALSE;
   A_3126_MXZ02MA.Mon5.Par.ParDelayChange := 0;
   A_3126_MXZ02MA.Mon5.Par.ParDelayTrue := 0;
   A_3126_MXZ02MA.Mon5.Par.ParDelayFalse := 0;
   A_3126_MXZ02MA.Mon5.Par.ParTimeoutTrue := 0;
   A_3126_MXZ02MA.Mon5.Par.ParTimeoutFalse := 0;
   A_3126_MXZ02MA.Mon5.Par.OutMonTime := 0;
   A_3126_MXZ02MA.Mon5.Par.OutTransitionTime := 0;
   A_3126_MXZ02MA.Mon5.Par.OutMonTrue := FALSE;
   A_3126_MXZ02MA.Mon5.Par.OutMonFalse := FALSE;
   A_3126_MXZ02MA.Mon5.Par.OutFlagFaultDev := FALSE;
   A_3126_MXZ02MA.Mon5.Par.OutDelayTime := 0;
   A_3126_MXZ02MA.Mon6.StCode := 0;
   A_3126_MXZ02MA.Mon6.InMonTrue := FALSE;
   A_3126_MXZ02MA.Mon6.InMonFalse := FALSE;
   A_3126_MXZ02MA.Mon6.InPreAlarmTrue := FALSE;
   A_3126_MXZ02MA.Mon6.InPreAlarmFalse := FALSE;
   A_3126_MXZ02MA.Mon6.InStopTrueTime := FALSE;
   A_3126_MXZ02MA.Mon6.InStopFalseTime := FALSE;
   A_3126_MXZ02MA.Mon6.InpTrue := FALSE;
   A_3126_MXZ02MA.Mon6.InpFaultDev := FALSE;
   A_3126_MXZ02MA.Mon6.CmdRstTrueTime := FALSE;
   A_3126_MXZ02MA.Mon6.CmdRstFalseTime := FALSE;
   A_3126_MXZ02MA.Mon6.CmdRunTimeoutTime := FALSE;
   A_3126_MXZ02MA.Mon6.CmdFaultReset := FALSE;
   A_3126_MXZ02MA.Mon6.InLocal := FALSE;
   A_3126_MXZ02MA.Mon6.spare0305 := FALSE;
   A_3126_MXZ02MA.Mon6.InReport := FALSE;
   A_3126_MXZ02MA.Mon6.OutTimeoutTime := FALSE;
   A_3126_MXZ02MA.Mon6.InHWStop := FALSE;
   A_3126_MXZ02MA.Mon6.InDPFault := FALSE;
   A_3126_MXZ02MA.Mon6.OutPreAlarmTrue := FALSE;
   A_3126_MXZ02MA.Mon6.OutPreAlarmFalse := FALSE;
   A_3126_MXZ02MA.Mon6.OutFlagPos := FALSE;
   A_3126_MXZ02MA.Mon6.OutFlagNeg := FALSE;
   A_3126_MXZ02MA.Mon6.OutpFaultReset := FALSE;
   A_3126_MXZ02MA.Mon6.OutTrue := FALSE;
   A_3126_MXZ02MA.Mon6.StFalse := FALSE;
   A_3126_MXZ02MA.Mon6.StCtoTrue := FALSE;
   A_3126_MXZ02MA.Mon6.StTrue := FALSE;
   A_3126_MXZ02MA.Mon6.StCtoFalse := FALSE;
   A_3126_MXZ02MA.Mon6.StFault := FALSE;
   A_3126_MXZ02MA.Mon6.OutAlarmNrLog := 0;
   A_3126_MXZ02MA.Mon6.Par.ParObjectNo := 0;
   A_3126_MXZ02MA.Mon6.Par.ParMsgType := 0;
   A_3126_MXZ02MA.Mon6.Par.ParHornCode := 0;
   A_3126_MXZ02MA.Mon6.Par.ParLogOff := FALSE;
   A_3126_MXZ02MA.Mon6.Par.spare0401 := FALSE;
   A_3126_MXZ02MA.Mon6.Par.Par2WorkingCond := FALSE;
   A_3126_MXZ02MA.Mon6.Par.ParFaultRetry := FALSE;
   A_3126_MXZ02MA.Mon6.Par.ParBinLevel := FALSE;
   A_3126_MXZ02MA.Mon6.Par.ParDelayChange := 0;
   A_3126_MXZ02MA.Mon6.Par.ParDelayTrue := 0;
   A_3126_MXZ02MA.Mon6.Par.ParDelayFalse := 0;
   A_3126_MXZ02MA.Mon6.Par.ParTimeoutTrue := 0;
   A_3126_MXZ02MA.Mon6.Par.ParTimeoutFalse := 0;
   A_3126_MXZ02MA.Mon6.Par.OutMonTime := 0;
   A_3126_MXZ02MA.Mon6.Par.OutTransitionTime := 0;
   A_3126_MXZ02MA.Mon6.Par.OutMonTrue := FALSE;
   A_3126_MXZ02MA.Mon6.Par.OutMonFalse := FALSE;
   A_3126_MXZ02MA.Mon6.Par.OutFlagFaultDev := FALSE;
   A_3126_MXZ02MA.Mon6.Par.OutDelayTime := 0;
   A_3126_MXZ02MA.A_3225_MXZ02.StCode := 0;
   A_3126_MXZ02MA.A_3225_MXZ02.InEnableRev := FALSE;
   A_3126_MXZ02MA.A_3225_MXZ02.InEnableFwd := FALSE;
   A_3126_MXZ02MA.A_3225_MXZ02.InSlow := FALSE;
   A_3126_MXZ02MA.A_3225_MXZ02.InpRunSlow := FALSE;
   A_3126_MXZ02MA.A_3225_MXZ02.InpRunFast := FALSE;
   A_3126_MXZ02MA.A_3225_MXZ02.InpRunRev := FALSE;
   A_3126_MXZ02MA.A_3225_MXZ02.InpRunFwd := FALSE;
   A_3126_MXZ02MA.A_3225_MXZ02.InpFaultDev := FALSE;
   A_3126_MXZ02MA.A_3225_MXZ02.CmdOff := FALSE;
   A_3126_MXZ02MA.A_3225_MXZ02.CmdOn := FALSE;
   A_3126_MXZ02MA.A_3225_MXZ02.CmdNext := FALSE;
   A_3126_MXZ02MA.A_3225_MXZ02.CmdFaultReset := FALSE;
   A_3126_MXZ02MA.A_3225_MXZ02.InLocal := FALSE;
   A_3126_MXZ02MA.A_3225_MXZ02.InManual := FALSE;
   A_3126_MXZ02MA.A_3225_MXZ02.InReport := FALSE;
   A_3126_MXZ02MA.A_3225_MXZ02.InSeqStop := FALSE;
   A_3126_MXZ02MA.A_3225_MXZ02.InHWStop := FALSE;
   A_3126_MXZ02MA.A_3225_MXZ02.InDPFault := FALSE;
   A_3126_MXZ02MA.A_3225_MXZ02.OutIdling := FALSE;
   A_3126_MXZ02MA.A_3225_MXZ02.OutpRunSlow := FALSE;
   A_3126_MXZ02MA.A_3225_MXZ02.OutpRunFast := FALSE;
   A_3126_MXZ02MA.A_3225_MXZ02.OutpRunRev := FALSE;
   A_3126_MXZ02MA.A_3225_MXZ02.OutpRunFwd := FALSE;
   A_3126_MXZ02MA.A_3225_MXZ02.OutpFaultReset := FALSE;
   A_3126_MXZ02MA.A_3225_MXZ02.StStopped := FALSE;
   A_3126_MXZ02MA.A_3225_MXZ02.StStarting := FALSE;
   A_3126_MXZ02MA.A_3225_MXZ02.StStartedFwd := FALSE;
   A_3126_MXZ02MA.A_3225_MXZ02.StStopping := FALSE;
   A_3126_MXZ02MA.A_3225_MXZ02.StFault := FALSE;
   A_3126_MXZ02MA.A_3225_MXZ02.StStartedRev := FALSE;
   A_3126_MXZ02MA.A_3225_MXZ02.InOutManSlow := FALSE;
   A_3126_MXZ02MA.A_3225_MXZ02.InOutManRev := FALSE;
   A_3126_MXZ02MA.A_3225_MXZ02.OutAlarmNrLog := 0;
   A_3126_MXZ02MA.A_3225_MXZ02.Par.ParObjectNo := 27133;
   A_3126_MXZ02MA.A_3225_MXZ02.Par.ParMsgType := 7053;
   A_3126_MXZ02MA.A_3225_MXZ02.Par.ParHornCode := 10;
   A_3126_MXZ02MA.A_3225_MXZ02.Par.ParLogOff := FALSE;
   A_3126_MXZ02MA.A_3225_MXZ02.Par.ParManual := TRUE;
   A_3126_MXZ02MA.A_3225_MXZ02.Par.ParRestartDelay := FALSE;
   A_3126_MXZ02MA.A_3225_MXZ02.Par.Par2Speed := FALSE;
   A_3126_MXZ02MA.A_3225_MXZ02.Par.ParHeavyStartup := FALSE;
   A_3126_MXZ02MA.A_3225_MXZ02.Par.spare45 := FALSE;
   A_3126_MXZ02MA.A_3225_MXZ02.Par.spare46 := FALSE;
   A_3126_MXZ02MA.A_3225_MXZ02.Par.OutEdgeFaultReset := FALSE;
   A_3126_MXZ02MA.A_3225_MXZ02.Par.OutDelayFault := FALSE;
   A_3126_MXZ02MA.A_3225_MXZ02.Par.OutFlagFaultDev := FALSE;
   A_3126_MXZ02MA.A_3225_MXZ02.Par.ParMonTime := 20;
   A_3126_MXZ02MA.A_3225_MXZ02.Par.ParStartingTime := 20;
   A_3126_MXZ02MA.A_3225_MXZ02.Par.ParStoppingTime := 0;
   A_3126_MXZ02MA.A_3225_MXZ02.Par.ParIdlingTime := 0;
   A_3126_MXZ02MA.A_3225_MXZ02.Par.ParDelayTime := 10;
   A_3126_MXZ02MA.A_3225_MXZ02.Par.OutMonTime := 0;
   A_3126_MXZ02MA.A_3225_MXZ02.Par.OutTransitionTime := 0;
   A_3126_MXZ02MA.A_3225_MXZ02.Par.OutDelayTime := 0;
   A_3126_MXZ02MA.A_3225_MXZ02.Par.InOutManPulseLen := 0;
END_DATA_BLOCK


